LIN {X 0,Y 639.897,Z 1293.567,A -85,B 0,C 180,E1 29787.314,E2 29787.314} C_VEL
LIN {X 0,Y 639.907,Z 1290.691,A -85,B 0,C 180,E1 29785.251,E2 29785.251} C_VEL
LIN {X 0,Y 639.948,Z 1285.814,A -85,B 0,C 180,E1 29783.091,E2 29783.091} C_VEL
LIN {X 0,Y 640.038,Z 1280.646,A -85,B 0,C 180,E1 29781.376,E2 29781.376} C_VEL
LIN {X 0,Y 640.175,Z 1274.233,A -85,B 0,C 180,E1 29779.654,E2 29779.654} C_VEL
LIN {X 0,Y 640.418,Z 1265.861,A -85,B 0,C 180,E1 29777.791,E2 29777.791} C_VEL
LIN {X 0,Y 640.846,Z 1254.401,A -85,B 0,C 180,E1 29775.68,E2 29775.68} C_VEL
LIN {X 0,Y 641.338,Z 1242.79,A -85,B 0,C 180,E1 29773.89,E2 29773.89} C_VEL
LIN {X 0,Y 641.901,Z 1231.865,A -85,B 0,C 180,E1 29772.412,E2 29772.412} C_VEL
LIN {X 0,Y 642.587,Z 1219.47,A -85,B 0,C 180,E1 29770.929,E2 29770.929} C_VEL
LIN {X 0,Y 643.506,Z 1204.493,A -85,B 0,C 180,E1 29769.348,E2 29769.348} C_VEL
LIN {X 0,Y 644.672,Z 1186.015,A -85,B 0,C 180,E1 29767.668,E2 29767.668} C_VEL
LIN {X 0,Y 645.836,Z 1168.25,A -85,B 0,C 180,E1 29766.265,E2 29766.265} C_VEL
LIN {X 0,Y 647.147,Z 1148.227,A -85,B 0,C 180,E1 29764.907,E2 29764.907} C_VEL
LIN {X 0,Y 648.4,Z 1127.933,A -85,B 0,C 180,E1 29763.733,E2 29763.733} C_VEL
LIN {X 0,Y 649.554,Z 1106.2,A -85,B 0,C 180,E1 29762.697,E2 29762.697} C_VEL
LIN {X 0,Y 650.662,Z 1083.667,A -85,B 0,C 180,E1 29761.802,E2 29761.802} C_VEL
LIN {X 0,Y 651.674,Z 1060.243,A -85,B 0,C 180,E1 29761.049,E2 29761.049} C_VEL
LIN {X 0,Y 652.617,Z 1036.441,A -85,B 0,C 180,E1 29760.454,E2 29760.454} C_VEL
LIN {X 0,Y 653.293,Z 1013.421,A -85,B 0,C 180,E1 29760.036,E2 29760.036} C_VEL
LIN {X 0,Y 654.171,Z 971.336,A -85,B 0,C 180,E1 29759.507,E2 29759.507} C_VEL
LIN {X 0,Y 659.659,Z 959.553,A -85,B 0,C 180,E1 29758.879,E2 29758.879} C_VEL
LIN {X 0,Y 664.536,Z 951.202,A -85,B 0,C 180,E1 29758.477,E2 29758.477} C_VEL
LIN {X 0,Y 670.603,Z 941.643,A -85,B 0,C 180,E1 29758.043,E2 29758.043} C_VEL
LIN {X 0,Y 679.475,Z 930.778,A -85,B 0,C 180,E1 29757.638,E2 29757.638} C_VEL
LIN {X 0,Y 692.272,Z 917.65,A -85,B 0,C 180,E1 29757.261,E2 29757.261} C_VEL
LIN {X 0,Y 701.55,Z 907.268,A -85,B 0,C 180,E1 29757.112,E2 29757.112} C_VEL
LIN {X 0,Y 709.193,Z 894.911,A -85,B 0,C 180,E1 29756.838,E2 29756.838} C_VEL
LIN {X 0,Y 716.952,Z 880.627,A -85,B 0,C 180,E1 29756.657,E2 29756.657} C_VEL
LIN {X 0,Y 714.524,Z 882.399,A -85,B 0,C 180,E1 29756.226,E2 29756.226} C_VEL
LIN {X 0,Y 710.853,Z 883.16,A -85,B 0,C 180,E1 29755.801,E2 29755.801} C_VEL
LIN {X 0,Y 705.825,Z 882.559,A -85,B 0,C 180,E1 29755.393,E2 29755.393} C_VEL
LIN {X 0,Y 694.35,Z 878.529,A -85,B 0,C 180,E1 29754.594,E2 29754.594} C_VEL
LIN {X 0,Y 684.4,Z 873.303,A -85,B 0,C 180,E1 29753.752,E2 29753.752} C_VEL
LIN {X 0,Y 675.328,Z 866.486,A -85,B 0,C 180,E1 29752.803,E2 29752.803} C_VEL
LIN {X 0,Y 667.782,Z 858.379,A -85,B 0,C 180,E1 29751.803,E2 29751.803} C_VEL
LIN {X 0,Y 661.627,Z 848.569,A -85,B 0,C 180,E1 29750.714,E2 29750.714} C_VEL
LIN {X 0,Y 657.041,Z 836.989,A -85,B 0,C 180,E1 29749.544,E2 29749.544} C_VEL
LIN {X 0,Y 654.419,Z 824.683,A -85,B 0,C 180,E1 29748.41,E2 29748.41} C_VEL
LIN {X 0,Y 653.38,Z 808.168,A -85,B 0,C 180,E1 29747.013,E2 29747.013} C_VEL
LIN {X 0,Y 655.589,Z 761.985,A -85,B 0,C 180,E1 29743.341,E2 29743.341} C_VEL
LIN {X 0,Y 657.511,Z 726.256,A -85,B 0,C 180,E1 29740.43,E2 29740.43} C_VEL
LIN {X 0,Y 659.372,Z 691.646,A -85,B 0,C 180,E1 29737.528,E2 29737.528} C_VEL
LIN {X 0,Y 661.157,Z 657.905,A -85,B 0,C 180,E1 29734.608,E2 29734.608} C_VEL
LIN {X 0,Y 661.133,Z 654.991,A -85,B 0,C 180,E1 29734.337,E2 29734.337} C_VEL
LIN {X 0,Y 652.452,Z 634.727,A -85,B 0,C 180,E1 29731.609,E2 29731.609} C_VEL
LIN {X 0,Y 645.602,Z 619.347,A -85,B 0,C 180,E1 29729.404,E2 29729.404} C_VEL
LIN {X 0,Y 642.088,Z 611.595,A -85,B 0,C 180,E1 29728.256,E2 29728.256} C_VEL
LIN {X 0,Y 640.822,Z 608.156,A -85,B 0,C 180,E1 29727.737,E2 29727.737} C_VEL
LIN {X 0,Y 640.824,Z 608.157,A -85,B 0,C 180,E1 29724.621,E2 29724.621} C_VEL
LIN {X 0,Y 640.829,Z 608.159,A -85,B 0,C 180,E1 29721.415,E2 29721.415} C_VEL
LIN {X 0,Y 640.828,Z 608.156,A -85,B 0,C 180,E1 29718.278,E2 29718.278} C_VEL
LIN {X 0,Y 640.832,Z 608.155,A -85,B 0,C 180,E1 29715.03,E2 29715.03} C_VEL
LIN {X 0,Y 640.836,Z 608.156,A -85,B 0,C 180,E1 29711.886,E2 29711.886} C_VEL
LIN {X 0,Y 640.828,Z 608.156,A -85,B 0,C 180,E1 29708.705,E2 29708.705} C_VEL
LIN {X 0,Y 640.835,Z 608.152,A -85,B 0,C 180,E1 29705.551,E2 29705.551} C_VEL
LIN {X 0,Y 640.822,Z 608.159,A -85,B 0,C 180,E1 29702.325,E2 29702.325} C_VEL
LIN {X 0,Y 640.833,Z 608.158,A -85,B 0,C 180,E1 29699.195,E2 29699.195} C_VEL
LIN {X 0,Y 640.819,Z 608.158,A -85,B 0,C 180,E1 29696.063,E2 29696.063} C_VEL
LIN {X 0,Y 640.828,Z 608.156,A -85,B 0,C 180,E1 29692.895,E2 29692.895} C_VEL
LIN {X 0,Y 640.816,Z 608.156,A -85,B 0,C 180,E1 29689.754,E2 29689.754} C_VEL
LIN {X 0,Y 640.823,Z 608.154,A -85,B 0,C 180,E1 29686.648,E2 29686.648} C_VEL
LIN {X 0,Y 640.817,Z 608.154,A -85,B 0,C 180,E1 29683.595,E2 29683.595} C_VEL
LIN {X 0,Y 640.823,Z 608.154,A -85,B 0,C 180,E1 29680.458,E2 29680.458} C_VEL
LIN {X 0,Y 640.816,Z 608.156,A -85,B 0,C 180,E1 29677.331,E2 29677.331} C_VEL
LIN {X 0,Y 640.818,Z 608.156,A -85,B 0,C 180,E1 29674.193,E2 29674.193} C_VEL
LIN {X 0,Y 640.816,Z 608.156,A -85,B 0,C 180,E1 29671.082,E2 29671.082} C_VEL
LIN {X 0,Y 640.816,Z 608.155,A -85,B 0,C 180,E1 29667.96,E2 29667.96} C_VEL
LIN {X 0,Y 640.815,Z 608.151,A -85,B 0,C 180,E1 29664.844,E2 29664.844} C_VEL
LIN {X 0,Y 640.816,Z 608.152,A -85,B 0,C 180,E1 29661.723,E2 29661.723} C_VEL
LIN {X 0,Y 640.817,Z 608.154,A -85,B 0,C 180,E1 29658.633,E2 29658.633} C_VEL
LIN {X 0,Y 640.817,Z 608.152,A -85,B 0,C 180,E1 29655.483,E2 29655.483} C_VEL
LIN {X 0,Y 640.832,Z 608.158,A -85,B 0,C 180,E1 29654.378,E2 29654.378} C_VEL
LIN {X 0,Y 639.852,Z 608.286,A -85,B 0,C 180,E1 29653.69,E2 29653.69} C_VEL
LIN {X 0,Y 633.444,Z 609.065,A -85,B 0,C 180,E1 29651.759,E2 29651.759} C_VEL
LIN {X 0,Y 632.89,Z 609.134,A -85,B 0,C 180,E1 29651.257,E2 29651.257} C_VEL
LIN {X 0,Y 632.886,Z 609.141,A -85,B 0,C 180,E1 29648.114,E2 29648.114} C_VEL
LIN {X 0,Y 632.892,Z 609.141,A -85,B 0,C 180,E1 29644.919,E2 29644.919} C_VEL
LIN {X 0,Y 632.906,Z 609.283,A -85,B 0,C 180,E1 29642.246,E2 29642.246} C_VEL
LIN {X 0,Y 640.506,Z 633.883,A -85,B 0,C 180,E1 29640.279,E2 29640.279} C_VEL
LIN {X 0,Y 639.937,Z 670.595,A -85,B 0,C 180,E1 29637.804,E2 29637.804} C_VEL
LIN {X 0,Y 638.884,Z 712.937,A -85,B 0,C 180,E1 29634.896,E2 29634.896} C_VEL
LIN {X 0,Y 637.709,Z 757.785,A -85,B 0,C 180,E1 29631.813,E2 29631.813} C_VEL
LIN {X 0,Y 636.616,Z 804.939,A -85,B 0,C 180,E1 29628.639,E2 29628.639} C_VEL
LIN {X 0,Y 636.165,Z 836.355,A -85,B 0,C 180,E1 29626.604,E2 29626.604} C_VEL
LIN {X 0,Y 636.961,Z 845.526,A -85,B 0,C 180,E1 29626.473,E2 29626.473} C_VEL
LIN {X 0,Y 635.944,Z 1005.419,A -85,B 0,C 180,E1 29624.624,E2 29624.624} C_VEL
LIN {X 0,Y 635.746,Z 1022.874,A -85,B 0,C 180,E1 29624.256,E2 29624.256} C_VEL
LIN {X 0,Y 635.419,Z 1039.147,A -85,B 0,C 180,E1 29623.744,E2 29623.744} C_VEL
LIN {X 0,Y 634.987,Z 1055.365,A -85,B 0,C 180,E1 29623.058,E2 29623.058} C_VEL
LIN {X 0,Y 634.509,Z 1070.531,A -85,B 0,C 180,E1 29622.235,E2 29622.235} C_VEL
LIN {X 0,Y 634.009,Z 1084.629,A -85,B 0,C 180,E1 29621.276,E2 29621.276} C_VEL
LIN {X 0,Y 633.52,Z 1097.632,A -85,B 0,C 180,E1 29620.18,E2 29620.18} C_VEL
LIN {X 0,Y 633.087,Z 1109.143,A -85,B 0,C 180,E1 29618.994,E2 29618.994} C_VEL
LIN {X 0,Y 632.73,Z 1119.243,A -85,B 0,C 180,E1 29617.718,E2 29617.718} C_VEL
LIN {X 0,Y 632.454,Z 1127.914,A -85,B 0,C 180,E1 29616.352,E2 29616.352} C_VEL
LIN {X 0,Y 632.266,Z 1135.129,A -85,B 0,C 180,E1 29614.898,E2 29614.898} C_VEL
LIN {X 0,Y 632.152,Z 1140.845,A -85,B 0,C 180,E1 29613.354,E2 29613.354} C_VEL
LIN {X 0,Y 632.086,Z 1144.759,A -85,B 0,C 180,E1 29611.812,E2 29611.812} C_VEL
LIN {X 0,Y 632.068,Z 1147.012,A -85,B 0,C 180,E1 29610.18,E2 29610.18} C_VEL
LIN {X 0,Y 632.054,Z 1147.461,A -85,B 0,C 180,E1 29608.548,E2 29608.548} C_VEL
LIN {X 0,Y 632.072,Z 1146.132,A -85,B 0,C 180,E1 29606.916,E2 29606.916} C_VEL
LIN {X 0,Y 632.113,Z 1143.147,A -85,B 0,C 180,E1 29605.372,E2 29605.372} C_VEL
LIN {X 0,Y 632.203,Z 1138.378,A -85,B 0,C 180,E1 29603.825,E2 29603.825} C_VEL
LIN {X 0,Y 632.352,Z 1131.721,A -85,B 0,C 180,E1 29602.275,E2 29602.275} C_VEL
LIN {X 0,Y 632.597,Z 1123.458,A -85,B 0,C 180,E1 29600.813,E2 29600.813} C_VEL
LIN {X 0,Y 632.926,Z 1113.551,A -85,B 0,C 180,E1 29599.439,E2 29599.439} C_VEL
LIN {X 0,Y 633.356,Z 1102.074,A -85,B 0,C 180,E1 29598.156,E2 29598.156} C_VEL
LIN {X 0,Y 633.841,Z 1089.419,A -85,B 0,C 180,E1 29597.008,E2 29597.008} C_VEL
LIN {X 0,Y 634.337,Z 1075.597,A -85,B 0,C 180,E1 29595.997,E2 29595.997} C_VEL
LIN {X 0,Y 634.847,Z 1060.153,A -85,B 0,C 180,E1 29595.089,E2 29595.089} C_VEL
LIN {X 0,Y 635.28,Z 1044.944,A -85,B 0,C 180,E1 29594.386,E2 29594.386} C_VEL
LIN {X 0,Y 635.649,Z 1028.193,A -85,B 0,C 180,E1 29593.804,E2 29593.804} C_VEL
LIN {X 0,Y 635.902,Z 1010.504,A -85,B 0,C 180,E1 29593.376,E2 29593.376} C_VEL
LIN {X 0,Y 636.039,Z 990.987,A -85,B 0,C 180,E1 29593.097,E2 29593.097} C_VEL
LIN {X 0,Y 636.768,Z 841.145,A -85,B 0,C 180,E1 29591.38,E2 29591.38} C_VEL
LIN {X 0,Y 636.079,Z 835.695,A -85,B 0,C 180,E1 29591.295,E2 29591.295} C_VEL
LIN {X 0,Y 637.03,Z 786.131,A -85,B 0,C 180,E1 29588.015,E2 29588.015} C_VEL
LIN {X 0,Y 638.19,Z 740.132,A -85,B 0,C 180,E1 29584.874,E2 29584.874} C_VEL
LIN {X 0,Y 639.395,Z 696.862,A -85,B 0,C 180,E1 29581.884,E2 29581.884} C_VEL
LIN {X 0,Y 640.369,Z 654.586,A -85,B 0,C 180,E1 29578.984,E2 29578.984} C_VEL
LIN {X 0,Y 640.439,Z 633.256,A -85,B 0,C 180,E1 29577.542,E2 29577.542} C_VEL
LIN {X 0,Y 632.885,Z 609.139,A -85,B 0,C 180,E1 29575.559,E2 29575.559} C_VEL
LIN {X 0,Y 632.882,Z 609.145,A -85,B 0,C 180,E1 29572.329,E2 29572.329} C_VEL
LIN {X 0,Y 632.896,Z 609.135,A -85,B 0,C 180,E1 29569.15,E2 29569.15} C_VEL
LIN {X 0,Y 632.877,Z 609.144,A -85,B 0,C 180,E1 29565.959,E2 29565.959} C_VEL
LIN {X 0,Y 632.876,Z 609.144,A -85,B 0,C 180,E1 29562.854,E2 29562.854} C_VEL
LIN {X 0,Y 632.89,Z 609.145,A -85,B 0,C 180,E1 29559.781,E2 29559.781} C_VEL
LIN {X 0,Y 632.879,Z 609.146,A -85,B 0,C 180,E1 29556.621,E2 29556.621} C_VEL
LIN {X 0,Y 632.891,Z 609.15,A -85,B 0,C 180,E1 29553.462,E2 29553.462} C_VEL
LIN {X 0,Y 632.915,Z 609.376,A -85,B 0,C 180,E1 29552.998,E2 29552.998} C_VEL
LIN {X 0,Y 634.657,Z 613.86,A -85,B 0,C 180,E1 29552.448,E2 29552.448} C_VEL
LIN {X 0,Y 644.095,Z 628.518,A -85,B 0,C 180,E1 29551.604,E2 29551.604} C_VEL
LIN {X 0,Y 650.556,Z 639.812,A -85,B 0,C 180,E1 29551.027,E2 29551.027} C_VEL
LIN {X 0,Y 648.075,Z 791.876,A -85,B 0,C 180,E1 29549.096,E2 29549.096} C_VEL
LIN {X 0,Y 646.526,Z 902.715,A -85,B 0,C 180,E1 29547.714,E2 29547.714} C_VEL
LIN {X 0,Y 645.796,Z 953.532,A -85,B 0,C 180,E1 29547.058,E2 29547.058} C_VEL
LIN {X 0,Y 645.049,Z 977.906,A -85,B 0,C 180,E1 29546.565,E2 29546.565} C_VEL
LIN {X 0,Y 644.199,Z 999.937,A -85,B 0,C 180,E1 29545.958,E2 29545.958} C_VEL
LIN {X 0,Y 643.14,Z 1022.537,A -85,B 0,C 180,E1 29545.169,E2 29545.169} C_VEL
LIN {X 0,Y 641.904,Z 1044.009,A -85,B 0,C 180,E1 29544.233,E2 29544.233} C_VEL
LIN {X 0,Y 640.848,Z 1061.28,A -85,B 0,C 180,E1 29543.348,E2 29543.348} C_VEL
LIN {X 0,Y 639.771,Z 1077.595,A -85,B 0,C 180,E1 29542.387,E2 29542.387} C_VEL
LIN {X 0,Y 638.664,Z 1093.449,A -85,B 0,C 180,E1 29541.324,E2 29541.324} C_VEL
LIN {X 0,Y 637.522,Z 1109.728,A -85,B 0,C 180,E1 29540.089,E2 29540.089} C_VEL
LIN {X 0,Y 636.21,Z 1128.852,A -85,B 0,C 180,E1 29538.415,E2 29538.415} C_VEL
LIN {X 0,Y 635.223,Z 1143.488,A -85,B 0,C 180,E1 29536.93,E2 29536.93} C_VEL
LIN {X 0,Y 634.46,Z 1155.662,A -85,B 0,C 180,E1 29535.54,E2 29535.54} C_VEL
LIN {X 0,Y 633.782,Z 1167.178,A -85,B 0,C 180,E1 29534.061,E2 29534.061} C_VEL
LIN {X 0,Y 633.229,Z 1177.944,A -85,B 0,C 180,E1 29532.494,E2 29532.494} C_VEL
LIN {X 0,Y 632.78,Z 1187.36,A -85,B 0,C 180,E1 29530.931,E2 29530.931} C_VEL
LIN {X 0,Y 632.476,Z 1195.561,A -85,B 0,C 180,E1 29529.372,E2 29529.372} C_VEL
LIN {X 0,Y 632.221,Z 1203.41,A -85,B 0,C 180,E1 29527.634,E2 29527.634} C_VEL
LIN {X 0,Y 632.047,Z 1210.905,A -85,B 0,C 180,E1 29525.629,E2 29525.629} C_VEL
LIN {X 0,Y 631.95,Z 1217.313,A -85,B 0,C 180,E1 29523.356,E2 29523.356} C_VEL
LIN {X 0,Y 631.916,Z 1221.027,A -85,B 0,C 180,E1 29521.541,E2 29521.541} C_VEL
LIN {X 0,Y 631.906,Z 1223.496,A -85,B 0,C 180,E1 29519.728,E2 29519.728} C_VEL
LIN {X 0,Y 631.908,Z 1224.737,A -85,B 0,C 180,E1 29517.914,E2 29517.914} C_VEL
LIN {X 0,Y 631.914,Z 1224.788,A -85,B 0,C 180,E1 29516.189,E2 29516.189} C_VEL
LIN {X 0,Y 631.912,Z 1223.741,A -85,B 0,C 180,E1 29514.436,E2 29514.436} C_VEL
LIN {X 0,Y 631.921,Z 1221.197,A -85,B 0,C 180,E1 29512.453,E2 29512.453} C_VEL
LIN {X 0,Y 631.966,Z 1216.378,A -85,B 0,C 180,E1 29510.161,E2 29510.161} C_VEL
LIN {X 0,Y 632.052,Z 1210.665,A -85,B 0,C 180,E1 29508.225,E2 29508.225} C_VEL
LIN {X 0,Y 632.205,Z 1204.172,A -85,B 0,C 180,E1 29506.463,E2 29506.463} C_VEL
LIN {X 0,Y 632.439,Z 1196.31,A -85,B 0,C 180,E1 29504.691,E2 29504.691} C_VEL
LIN {X 0,Y 632.785,Z 1187.497,A -85,B 0,C 180,E1 29503.003,E2 29503.003} C_VEL
LIN {X 0,Y 633.295,Z 1176.659,A -85,B 0,C 180,E1 29501.211,E2 29501.211} C_VEL
LIN {X 0,Y 634.06,Z 1162.49,A -85,B 0,C 180,E1 29499.218,E2 29499.218} C_VEL
LIN {X 0,Y 634.861,Z 1149.049,A -85,B 0,C 180,E1 29497.595,E2 29497.595} C_VEL
LIN {X 0,Y 635.713,Z 1136.053,A -85,B 0,C 180,E1 29496.206,E2 29496.206} C_VEL
LIN {X 0,Y 636.625,Z 1122.428,A -85,B 0,C 180,E1 29494.908,E2 29494.908} C_VEL
LIN {X 0,Y 637.619,Z 1108.234,A -85,B 0,C 180,E1 29493.704,E2 29493.704} C_VEL
LIN {X 0,Y 638.659,Z 1093.556,A -85,B 0,C 180,E1 29492.594,E2 29492.594} C_VEL
LIN {X 0,Y 639.621,Z 1079.005,A -85,B 0,C 180,E1 29491.626,E2 29491.626} C_VEL
LIN {X 0,Y 640.712,Z 1061.526,A -85,B 0,C 180,E1 29490.606,E2 29490.606} C_VEL
LIN {X 0,Y 641.904,Z 1039.745,A -85,B 0,C 180,E1 29489.534,E2 29489.534} C_VEL
LIN {X 0,Y 642.868,Z 1018.864,A -85,B 0,C 180,E1 29488.702,E2 29488.702} C_VEL
LIN {X 0,Y 643.612,Z 999.264,A -85,B 0,C 180,E1 29488.058,E2 29488.058} C_VEL
LIN {X 0,Y 644.271,Z 976.224,A -85,B 0,C 180,E1 29487.472,E2 29487.472} C_VEL
LIN {X 0,Y 644.765,Z 952.724,A -85,B 0,C 180,E1 29487.047,E2 29487.047} C_VEL
LIN {X 0,Y 645.24,Z 868.019,A -85,B 0,C 180,E1 29486.099,E2 29486.099} C_VEL
LIN {X 0,Y 646.392,Z 666.407,A -85,B 0,C 180,E1 29483.836,E2 29483.836} C_VEL
LIN {X 0,Y 646.514,Z 638.485,A -85,B 0,C 180,E1 29483.499,E2 29483.499} C_VEL
LIN {X 0,Y 643.79,Z 635.766,A -85,B 0,C 180,E1 29483.341,E2 29483.341} C_VEL
LIN {X 0,Y 644,Z 636.198,A -85,B 0,C 180,E1 29482.172,E2 29482.172} C_VEL
LIN {X 0,Y 644.603,Z 638.016,A -85,B 0,C 180,E1 29481.195,E2 29481.195} C_VEL
LIN {X 0,Y 645.736,Z 641.08,A -85,B 0,C 180,E1 29480.178,E2 29480.178} C_VEL
LIN {X 0,Y 645.925,Z 642.037,A -85,B 0,C 180,E1 29479.951,E2 29479.951} C_VEL
LIN {X 0,Y 641.41,Z 653.382,A -85,B 0,C 180,E1 29478.712,E2 29478.712} C_VEL
LIN {X 0,Y 638.172,Z 666.32,A -85,B 0,C 180,E1 29477.523,E2 29477.523} C_VEL
LIN {X 0,Y 635.905,Z 681.652,A -85,B 0,C 180,E1 29476.328,E2 29476.328} C_VEL
LIN {X 0,Y 634.23,Z 702.463,A -85,B 0,C 180,E1 29474.935,E2 29474.935} C_VEL
LIN {X 0,Y 633.019,Z 734.797,A -85,B 0,C 180,E1 29473.03,E2 29473.03} C_VEL
LIN {X 0,Y 632.986,Z 773.811,A -85,B 0,C 180,E1 29470.88,E2 29470.88} C_VEL
LIN {X 0,Y 634.85,Z 794.261,A -85,B 0,C 180,E1 29469.752,E2 29469.752} C_VEL
LIN {X 0,Y 638.194,Z 811.119,A -85,B 0,C 180,E1 29468.808,E2 29468.808} C_VEL
LIN {X 0,Y 643.087,Z 825.935,A -85,B 0,C 180,E1 29467.973,E2 29467.973} C_VEL
LIN {X 0,Y 649.932,Z 840.295,A -85,B 0,C 180,E1 29467.163,E2 29467.163} C_VEL
LIN {X 0,Y 657.821,Z 852.497,A -85,B 0,C 180,E1 29466.478,E2 29466.478} C_VEL
LIN {X 0,Y 667.384,Z 863.872,A -85,B 0,C 180,E1 29465.851,E2 29465.851} C_VEL
LIN {X 0,Y 678.649,Z 874.385,A -85,B 0,C 180,E1 29465.29,E2 29465.29} C_VEL
LIN {X 0,Y 690.663,Z 883.187,A -85,B 0,C 180,E1 29464.829,E2 29464.829} C_VEL
LIN {X 0,Y 697.221,Z 887.009,A -85,B 0,C 180,E1 29464.595,E2 29464.595} C_VEL
LIN {X 0,Y 702.925,Z 889.045,A -85,B 0,C 180,E1 29464.285,E2 29464.285} C_VEL
LIN {X 0,Y 707.445,Z 889.627,A -85,B 0,C 180,E1 29463.936,E2 29463.936} C_VEL
LIN {X 0,Y 708.595,Z 889.733,A -85,B 0,C 180,E1 29463.813,E2 29463.813} C_VEL
LIN {X 0,Y 699.671,Z 901.616,A -85,B 0,C 180,E1 29463.529,E2 29463.529} C_VEL
LIN {X 0,Y 696.631,Z 905.632,A -85,B 0,C 180,E1 29463.398,E2 29463.398} C_VEL
LIN {X 0,Y 686.664,Z 914.581,A -85,B 0,C 180,E1 29463.144,E2 29463.144} C_VEL
LIN {X 0,Y 675.161,Z 924.295,A -85,B 0,C 180,E1 29462.672,E2 29462.672} C_VEL
LIN {X 0,Y 665.009,Z 934.556,A -85,B 0,C 180,E1 29462.109,E2 29462.109} C_VEL
LIN {X 0,Y 657.922,Z 944.123,A -85,B 0,C 180,E1 29461.572,E2 29461.572} C_VEL
LIN {X 0,Y 649.022,Z 959.216,A -85,B 0,C 180,E1 29460.712,E2 29460.712} C_VEL
LIN {X 0,Y 646.755,Z 964.415,A -85,B 0,C 180,E1 29460.447,E2 29460.447} C_VEL
LIN {X 0,Y 644.912,Z 973.272,A -85,B 0,C 180,E1 29460.398,E2 29460.398} C_VEL
LIN {X 0,Y 644.423,Z 1012.046,A -85,B 0,C 180,E1 29459.935,E2 29459.935} C_VEL
LIN {X 0,Y 643.83,Z 1038.212,A -85,B 0,C 180,E1 29459.462,E2 29459.462} C_VEL
LIN {X 0,Y 643.11,Z 1062.478,A -85,B 0,C 180,E1 29458.87,E2 29458.87} C_VEL
LIN {X 0,Y 642.378,Z 1085.145,A -85,B 0,C 180,E1 29458.177,E2 29458.177} C_VEL
LIN {X 0,Y 641.485,Z 1108.187,A -85,B 0,C 180,E1 29457.318,E2 29457.318} C_VEL
LIN {X 0,Y 640.506,Z 1130.491,A -85,B 0,C 180,E1 29456.319,E2 29456.319} C_VEL
LIN {X 0,Y 639.636,Z 1148.325,A -85,B 0,C 180,E1 29455.362,E2 29455.362} C_VEL
LIN {X 0,Y 638.63,Z 1164.294,A -85,B 0,C 180,E1 29454.317,E2 29454.317} C_VEL
LIN {X 0,Y 637.434,Z 1180.844,A -85,B 0,C 180,E1 29453.041,E2 29453.041} C_VEL
LIN {X 0,Y 636.455,Z 1195.131,A -85,B 0,C 180,E1 29451.8,E2 29451.8} C_VEL
LIN {X 0,Y 635.575,Z 1208.117,A -85,B 0,C 180,E1 29450.539,E2 29450.539} C_VEL
LIN {X 0,Y 634.734,Z 1221.071,A -85,B 0,C 180,E1 29449.128,E2 29449.128} C_VEL
LIN {X 0,Y 634.009,Z 1233.284,A -85,B 0,C 180,E1 29447.627,E2 29447.627} C_VEL
LIN {X 0,Y 633.349,Z 1245.331,A -85,B 0,C 180,E1 29445.945,E2 29445.945} C_VEL
LIN {X 0,Y 632.753,Z 1258.357,A -85,B 0,C 180,E1 29443.806,E2 29443.806} C_VEL
LIN {X 0,Y 632.418,Z 1267.357,A -85,B 0,C 180,E1 29442.047,E2 29442.047} C_VEL
LIN {X 0,Y 632.181,Z 1274.952,A -85,B 0,C 180,E1 29440.297,E2 29440.297} C_VEL
LIN {X 0,Y 632.044,Z 1281.234,A -85,B 0,C 180,E1 29438.553,E2 29438.553} C_VEL
LIN {X 0,Y 631.951,Z 1287.265,A -85,B 0,C 180,E1 29436.451,E2 29436.451} C_VEL
LIN {X 0,Y 631.913,Z 1291.566,A -85,B 0,C 180,E1 29434.266,E2 29434.266} C_VEL
LIN {X 0,Y 631.901,Z 1293.89,A -85,B 0,C 180,E1 29432.359,E2 29432.359} C_VEL
LIN {X 0,Y 631.893,Z 1294.865,A -85,B 0,C 180,E1 29430.545,E2 29430.545} C_VEL
LIN {X 0,Y 631.892,Z 1294.559,A -85,B 0,C 180,E1 29428.46,E2 29428.46} C_VEL
LIN {X 0,Y 631.9,Z 1292.387,A -85,B 0,C 180,E1 29426.282,E2 29426.282} C_VEL
LIN {X 0,Y 631.921,Z 1289.037,A -85,B 0,C 180,E1 29424.371,E2 29424.371} C_VEL
LIN {X 0,Y 631.991,Z 1284.804,A -85,B 0,C 180,E1 29422.639,E2 29422.639} C_VEL
LIN {X 0,Y 632.068,Z 1279.397,A -85,B 0,C 180,E1 29420.899,E2 29420.899} C_VEL
LIN {X 0,Y 632.276,Z 1271.619,A -85,B 0,C 180,E1 29418.877,E2 29418.877} C_VEL
LIN {X 0,Y 632.632,Z 1261.37,A -85,B 0,C 180,E1 29416.753,E2 29416.753} C_VEL
LIN {X 0,Y 633.026,Z 1251.836,A -85,B 0,C 180,E1 29415.082,E2 29415.082} C_VEL
LIN {X 0,Y 633.521,Z 1242.136,A -85,B 0,C 180,E1 29413.591,E2 29413.591} C_VEL
LIN {X 0,Y 634.13,Z 1231.127,A -85,B 0,C 180,E1 29412.094,E2 29412.094} C_VEL
LIN {X 0,Y 634.895,Z 1218.644,A -85,B 0,C 180,E1 29410.593,E2 29410.593} C_VEL
LIN {X 0,Y 635.991,Z 1202.167,A -85,B 0,C 180,E1 29408.851,E2 29408.851} C_VEL
LIN {X 0,Y 637.169,Z 1184.867,A -85,B 0,C 180,E1 29407.293,E2 29407.293} C_VEL
LIN {X 0,Y 638.369,Z 1167.956,A -85,B 0,C 180,E1 29405.947,E2 29405.947} C_VEL
LIN {X 0,Y 639.448,Z 1151.512,A -85,B 0,C 180,E1 29404.831,E2 29404.831} C_VEL
LIN {X 0,Y 640.748,Z 1130.264,A -85,B 0,C 180,E1 29403.595,E2 29403.595} C_VEL
LIN {X 0,Y 642.017,Z 1108.247,A -85,B 0,C 180,E1 29402.506,E2 29402.506} C_VEL
LIN {X 0,Y 643.29,Z 1085.07,A -85,B 0,C 180,E1 29401.553,E2 29401.553} C_VEL
LIN {X 0,Y 644.468,Z 1060.94,A -85,B 0,C 180,E1 29400.748,E2 29400.748} C_VEL
LIN {X 0,Y 645.547,Z 1036.841,A -85,B 0,C 180,E1 29400.124,E2 29400.124} C_VEL
LIN {X 0,Y 646.347,Z 1013.026,A -85,B 0,C 180,E1 29399.678,E2 29399.678} C_VEL
LIN {X 0,Y 647.327,Z 970.69,A -85,B 0,C 180,E1 29399.145,E2 29399.145} C_VEL
LIN {X 0,Y 647.893,Z 968.867,A -85,B 0,C 180,E1 29399.077,E2 29399.077} C_VEL
LIN {X 0,Y 653.309,Z 957.677,A -85,B 0,C 180,E1 29398.484,E2 29398.484} C_VEL
LIN {X 0,Y 662.94,Z 941.728,A -85,B 0,C 180,E1 29397.731,E2 29397.731} C_VEL
LIN {X 0,Y 671.242,Z 931.043,A -85,B 0,C 180,E1 29397.313,E2 29397.313} C_VEL
LIN {X 0,Y 683.251,Z 918.336,A -85,B 0,C 180,E1 29396.919,E2 29396.919} C_VEL
LIN {X 0,Y 697.669,Z 904.35,A -85,B 0,C 180,E1 29396.562,E2 29396.562} C_VEL
LIN {X 0,Y 706.24,Z 892.92,A -85,B 0,C 180,E1 29396.248,E2 29396.248} C_VEL
LIN {X 0,Y 708.556,Z 889.584,A -85,B 0,C 180,E1 29396.169,E2 29396.169} C_VEL
LIN {X 0,Y 703.814,Z 889.238,A -85,B 0,C 180,E1 29395.775,E2 29395.775} C_VEL
LIN {X 0,Y 691.427,Z 885.234,A -85,B 0,C 180,E1 29394.936,E2 29394.936} C_VEL
LIN {X 0,Y 680.59,Z 879.9,A -85,B 0,C 180,E1 29394.048,E2 29394.048} C_VEL
LIN {X 0,Y 670.686,Z 872.883,A -85,B 0,C 180,E1 29393.044,E2 29393.044} C_VEL
LIN {X 0,Y 662.472,Z 864.527,A -85,B 0,C 180,E1 29391.987,E2 29391.987} C_VEL
LIN {X 0,Y 656.416,Z 855.68,A -85,B 0,C 180,E1 29390.974,E2 29390.974} C_VEL
LIN {X 0,Y 651.308,Z 844.456,A -85,B 0,C 180,E1 29389.798,E2 29389.798} C_VEL
LIN {X 0,Y 647.974,Z 831.785,A -85,B 0,C 180,E1 29388.586,E2 29388.586} C_VEL
LIN {X 0,Y 646.455,Z 816.908,A -85,B 0,C 180,E1 29387.282,E2 29387.282} C_VEL
LIN {X 0,Y 646.864,Z 797.203,A -85,B 0,C 180,E1 29385.681,E2 29385.681} C_VEL
LIN {X 0,Y 648.952,Z 759.88,A -85,B 0,C 180,E1 29382.683,E2 29382.683} C_VEL
LIN {X 0,Y 650.979,Z 724.578,A -85,B 0,C 180,E1 29379.778,E2 29379.778} C_VEL
LIN {X 0,Y 652.917,Z 690.527,A -85,B 0,C 180,E1 29376.893,E2 29376.893} C_VEL
LIN {X 0,Y 654.678,Z 659.351,A -85,B 0,C 180,E1 29374.169,E2 29374.169} C_VEL
LIN {X 0,Y 646.087,Z 639.23,A -85,B 0,C 180,E1 29371.436,E2 29371.436} C_VEL
LIN {X 0,Y 638.251,Z 621.301,A -85,B 0,C 180,E1 29368.85,E2 29368.85} C_VEL
LIN {X 0,Y 634.191,Z 612.62,A -85,B 0,C 180,E1 29367.514,E2 29367.514} C_VEL
LIN {X 0,Y 632.878,Z 609.148,A -85,B 0,C 180,E1 29366.964,E2 29366.964} C_VEL
LIN {X 0,Y 632.874,Z 609.148,A -85,B 0,C 180,E1 29363.831,E2 29363.831} C_VEL
LIN {X 0,Y 632.882,Z 609.144,A -85,B 0,C 180,E1 29360.823,E2 29360.823} C_VEL
LIN {X 0,Y 632.875,Z 609.147,A -85,B 0,C 180,E1 29357.701,E2 29357.701} C_VEL
LIN {X 0,Y 632.892,Z 609.145,A -85,B 0,C 180,E1 29354.642,E2 29354.642} C_VEL
LIN {X 0,Y 632.881,Z 609.146,A -85,B 0,C 180,E1 29351.482,E2 29351.482} C_VEL
LIN {X 0,Y 632.894,Z 609.143,A -85,B 0,C 180,E1 29348.357,E2 29348.357} C_VEL
LIN {X 0,Y 632.89,Z 609.147,A -85,B 0,C 180,E1 29345.258,E2 29345.258} C_VEL
LIN {X 0,Y 632.89,Z 609.147,A -85,B 0,C 180,E1 29342.082,E2 29342.082} C_VEL
LIN {X 0,Y 632.891,Z 609.144,A -85,B 0,C 180,E1 29338.914,E2 29338.914} C_VEL
LIN {X 0,Y 632.888,Z 609.144,A -85,B 0,C 180,E1 29335.742,E2 29335.742} C_VEL
LIN {X 0,Y 632.896,Z 609.143,A -85,B 0,C 180,E1 29332.556,E2 29332.556} C_VEL
LIN {X 0,Y 632.89,Z 609.144,A -85,B 0,C 180,E1 29329.348,E2 29329.348} C_VEL
LIN {X 0,Y 632.895,Z 609.143,A -85,B 0,C 180,E1 29326.198,E2 29326.198} C_VEL
LIN {X 0,Y 632.89,Z 609.144,A -85,B 0,C 180,E1 29323.006,E2 29323.006} C_VEL
LIN {X 0,Y 632.892,Z 609.144,A -85,B 0,C 180,E1 29319.786,E2 29319.786} C_VEL
LIN {X 0,Y 632.89,Z 609.143,A -85,B 0,C 180,E1 29316.617,E2 29316.617} C_VEL
LIN {X 0,Y 632.889,Z 609.143,A -85,B 0,C 180,E1 29313.442,E2 29313.442} C_VEL
LIN {X 0,Y 632.891,Z 609.146,A -85,B 0,C 180,E1 29310.259,E2 29310.259} C_VEL
LIN {X 0,Y 632.891,Z 609.149,A -85,B 0,C 180,E1 29307.079,E2 29307.079} C_VEL
LIN {X 0,Y 632.886,Z 609.147,A -85,B 0,C 180,E1 29303.893,E2 29303.893} C_VEL
LIN {X 0,Y 632.894,Z 609.144,A -85,B 0,C 180,E1 29300.724,E2 29300.724} C_VEL
LIN {X 0,Y 632.891,Z 609.134,A -85,B 0,C 180,E1 29297.676,E2 29297.676} C_VEL
LIN {X 0,Y 632.892,Z 609.144,A -85,B 0,C 180,E1 29294.542,E2 29294.542} C_VEL
LIN {X 0,Y 632.895,Z 609.133,A -85,B 0,C 180,E1 29291.327,E2 29291.327} C_VEL
LIN {X 0,Y 632.89,Z 609.134,A -85,B 0,C 180,E1 29291.257,E2 29291.257} C_VEL
LIN {X 0,Y 631.871,Z 609.27,A -85,B 0,C 180,E1 29290.559,E2 29290.559} C_VEL
LIN {X 0,Y 625.46,Z 610.073,A -85,B 0,C 180,E1 29288.604,E2 29288.604} C_VEL
LIN {X 0,Y 624.948,Z 610.129,A -85,B 0,C 180,E1 29288.095,E2 29288.095} C_VEL
LIN {X 0,Y 624.953,Z 610.13,A -85,B 0,C 180,E1 29284.942,E2 29284.942} C_VEL
LIN {X 0,Y 624.945,Z 610.183,A -85,B 0,C 180,E1 29282.572,E2 29282.572} C_VEL
LIN {X 0,Y 633.076,Z 636.237,A -85,B 0,C 180,E1 29280.462,E2 29280.462} C_VEL
LIN {X 0,Y 632.487,Z 671.625,A -85,B 0,C 180,E1 29278.058,E2 29278.058} C_VEL
LIN {X 0,Y 631.415,Z 712.92,A -85,B 0,C 180,E1 29275.211,E2 29275.211} C_VEL
LIN {X 0,Y 630.182,Z 757.346,A -85,B 0,C 180,E1 29272.136,E2 29272.136} C_VEL
LIN {X 0,Y 629.033,Z 804.838,A -85,B 0,C 180,E1 29268.92,E2 29268.92} C_VEL
LIN {X 0,Y 628.541,Z 837.035,A -85,B 0,C 180,E1 29266.826,E2 29266.826} C_VEL
LIN {X 0,Y 629.358,Z 846.117,A -85,B 0,C 180,E1 29266.694,E2 29266.694} C_VEL
LIN {X 0,Y 628.274,Z 1006.384,A -85,B 0,C 180,E1 29264.818,E2 29264.818} C_VEL
LIN {X 0,Y 628.071,Z 1023.826,A -85,B 0,C 180,E1 29264.446,E2 29264.446} C_VEL
LIN {X 0,Y 627.723,Z 1040.405,A -85,B 0,C 180,E1 29263.916,E2 29263.916} C_VEL
LIN {X 0,Y 627.274,Z 1056.561,A -85,B 0,C 180,E1 29263.222,E2 29263.222} C_VEL
LIN {X 0,Y 626.771,Z 1071.683,A -85,B 0,C 180,E1 29262.389,E2 29262.389} C_VEL
LIN {X 0,Y 626.241,Z 1085.731,A -85,B 0,C 180,E1 29261.418,E2 29261.418} C_VEL
LIN {X 0,Y 625.719,Z 1098.711,A -85,B 0,C 180,E1 29260.309,E2 29260.309} C_VEL
LIN {X 0,Y 625.255,Z 1110.202,A -85,B 0,C 180,E1 29259.108,E2 29259.108} C_VEL
LIN {X 0,Y 624.869,Z 1120.286,A -85,B 0,C 180,E1 29257.816,E2 29257.816} C_VEL
LIN {X 0,Y 624.567,Z 1128.934,A -85,B 0,C 180,E1 29256.433,E2 29256.433} C_VEL
LIN {X 0,Y 624.357,Z 1136.135,A -85,B 0,C 180,E1 29254.96,E2 29254.96} C_VEL
LIN {X 0,Y 624.226,Z 1141.839,A -85,B 0,C 180,E1 29253.396,E2 29253.396} C_VEL
LIN {X 0,Y 624.15,Z 1145.739,A -85,B 0,C 180,E1 29251.835,E2 29251.835} C_VEL
LIN {X 0,Y 624.126,Z 1147.974,A -85,B 0,C 180,E1 29250.182,E2 29250.182} C_VEL
LIN {X 0,Y 624.111,Z 1148.411,A -85,B 0,C 180,E1 29248.53,E2 29248.53} C_VEL
LIN {X 0,Y 624.133,Z 1147.07,A -85,B 0,C 180,E1 29246.876,E2 29246.876} C_VEL
LIN {X 0,Y 624.183,Z 1144.065,A -85,B 0,C 180,E1 29245.313,E2 29245.313} C_VEL
LIN {X 0,Y 624.287,Z 1139.283,A -85,B 0,C 180,E1 29243.746,E2 29243.746} C_VEL
LIN {X 0,Y 624.457,Z 1132.61,A -85,B 0,C 180,E1 29242.176,E2 29242.176} C_VEL
LIN {X 0,Y 624.729,Z 1124.321,A -85,B 0,C 180,E1 29240.696,E2 29240.696} C_VEL
LIN {X 0,Y 625.09,Z 1114.393,A -85,B 0,C 180,E1 29239.306,E2 29239.306} C_VEL
LIN {X 0,Y 625.557,Z 1102.891,A -85,B 0,C 180,E1 29238.006,E2 29238.006} C_VEL
LIN {X 0,Y 626.075,Z 1090.191,A -85,B 0,C 180,E1 29236.844,E2 29236.844} C_VEL
LIN {X 0,Y 626.604,Z 1076.329,A -85,B 0,C 180,E1 29235.82,E2 29235.82} C_VEL
LIN {X 0,Y 627.121,Z 1061.464,A -85,B 0,C 180,E1 29234.935,E2 29234.935} C_VEL
LIN {X 0,Y 627.599,Z 1045.541,A -85,B 0,C 180,E1 29234.19,E2 29234.19} C_VEL
LIN {X 0,Y 627.978,Z 1028.723,A -85,B 0,C 180,E1 29233.603,E2 29233.603} C_VEL
LIN {X 0,Y 628.24,Z 1010.693,A -85,B 0,C 180,E1 29233.168,E2 29233.168} C_VEL
LIN {X 0,Y 628.374,Z 990.455,A -85,B 0,C 180,E1 29232.883,E2 29232.883} C_VEL
LIN {X 0,Y 629.154,Z 841.795,A -85,B 0,C 180,E1 29231.158,E2 29231.158} C_VEL
LIN {X 0,Y 628.484,Z 836.326,A -85,B 0,C 180,E1 29231.06,E2 29231.06} C_VEL
LIN {X 0,Y 629.458,Z 786.974,A -85,B 0,C 180,E1 29227.785,E2 29227.785} C_VEL
LIN {X 0,Y 630.691,Z 740.753,A -85,B 0,C 180,E1 29224.61,E2 29224.61} C_VEL
LIN {X 0,Y 631.946,Z 697.629,A -85,B 0,C 180,E1 29221.61,E2 29221.61} C_VEL
LIN {X 0,Y 632.975,Z 655.66,A -85,B 0,C 180,E1 29218.716,E2 29218.716} C_VEL
LIN {X 0,Y 633.245,Z 636.49,A -85,B 0,C 180,E1 29217.422,E2 29217.422} C_VEL
LIN {X 0,Y 625.703,Z 612.671,A -85,B 0,C 180,E1 29215.466,E2 29215.466} C_VEL
LIN {X 0,Y 624.943,Z 610.133,A -85,B 0,C 180,E1 29215.25,E2 29215.25} C_VEL
LIN {X 0,Y 624.935,Z 610.134,A -85,B 0,C 180,E1 29212.073,E2 29212.073} C_VEL
LIN {X 0,Y 624.95,Z 610.127,A -85,B 0,C 180,E1 29209.005,E2 29209.005} C_VEL
LIN {X 0,Y 624.936,Z 610.133,A -85,B 0,C 180,E1 29205.893,E2 29205.893} C_VEL
LIN {X 0,Y 624.937,Z 610.133,A -85,B 0,C 180,E1 29202.843,E2 29202.843} C_VEL
LIN {X 0,Y 624.952,Z 610.134,A -85,B 0,C 180,E1 29199.791,E2 29199.791} C_VEL
LIN {X 0,Y 624.941,Z 610.135,A -85,B 0,C 180,E1 29196.641,E2 29196.641} C_VEL
LIN {X 0,Y 624.984,Z 610.325,A -85,B 0,C 180,E1 29193.611,E2 29193.611} C_VEL
LIN {X 0,Y 627.037,Z 615.647,A -85,B 0,C 180,E1 29192.947,E2 29192.947} C_VEL
LIN {X 0,Y 638.063,Z 632.404,A -85,B 0,C 180,E1 29191.943,E2 29191.943} C_VEL
LIN {X 0,Y 643.99,Z 642.733,A -85,B 0,C 180,E1 29191.403,E2 29191.403} C_VEL
LIN {X 0,Y 639.965,Z 867.434,A -85,B 0,C 180,E1 29188.491,E2 29188.491} C_VEL
LIN {X 0,Y 638.749,Z 951.649,A -85,B 0,C 180,E1 29187.422,E2 29187.422} C_VEL
LIN {X 0,Y 638.015,Z 976.275,A -85,B 0,C 180,E1 29186.939,E2 29186.939} C_VEL
LIN {X 0,Y 637.108,Z 998.971,A -85,B 0,C 180,E1 29186.324,E2 29186.324} C_VEL
LIN {X 0,Y 636.084,Z 1020.1,A -85,B 0,C 180,E1 29185.59,E2 29185.59} C_VEL
LIN {X 0,Y 634.745,Z 1042.604,A -85,B 0,C 180,E1 29184.629,E2 29184.629} C_VEL
LIN {X 0,Y 633.504,Z 1061.927,A -85,B 0,C 180,E1 29183.635,E2 29183.635} C_VEL
LIN {X 0,Y 632.192,Z 1080.752,A -85,B 0,C 180,E1 29182.504,E2 29182.504} C_VEL
LIN {X 0,Y 630.605,Z 1102.034,A -85,B 0,C 180,E1 29180.999,E2 29180.999} C_VEL
LIN {X 0,Y 629.391,Z 1117.968,A -85,B 0,C 180,E1 29179.682,E2 29179.682} C_VEL
LIN {X 0,Y 628.32,Z 1132.088,A -85,B 0,C 180,E1 29178.366,E2 29178.366} C_VEL
LIN {X 0,Y 627.428,Z 1144.695,A -85,B 0,C 180,E1 29177.051,E2 29177.051} C_VEL
LIN {X 0,Y 626.617,Z 1156.737,A -85,B 0,C 180,E1 29175.645,E2 29175.645} C_VEL
LIN {X 0,Y 625.942,Z 1167.462,A -85,B 0,C 180,E1 29174.241,E2 29174.241} C_VEL
LIN {X 0,Y 625.334,Z 1178.195,A -85,B 0,C 180,E1 29172.654,E2 29172.654} C_VEL
LIN {X 0,Y 624.855,Z 1187.581,A -85,B 0,C 180,E1 29171.071,E2 29171.071} C_VEL
LIN {X 0,Y 624.521,Z 1195.752,A -85,B 0,C 180,E1 29169.492,E2 29169.492} C_VEL
LIN {X 0,Y 624.245,Z 1203.57,A -85,B 0,C 180,E1 29167.733,E2 29167.733} C_VEL
LIN {X 0,Y 624.059,Z 1211.037,A -85,B 0,C 180,E1 29165.701,E2 29165.701} C_VEL
LIN {X 0,Y 623.954,Z 1217.195,A -85,B 0,C 180,E1 29163.491,E2 29163.491} C_VEL
LIN {X 0,Y 623.917,Z 1221.084,A -85,B 0,C 180,E1 29161.561,E2 29161.561} C_VEL
LIN {X 0,Y 623.907,Z 1223.528,A -85,B 0,C 180,E1 29159.725,E2 29159.725} C_VEL
LIN {X 0,Y 623.91,Z 1224.714,A -85,B 0,C 180,E1 29157.979,E2 29157.979} C_VEL
LIN {X 0,Y 623.914,Z 1224.799,A -85,B 0,C 180,E1 29156.233,E2 29156.233} C_VEL
LIN {X 0,Y 623.911,Z 1223.804,A -85,B 0,C 180,E1 29154.482,E2 29154.482} C_VEL
LIN {X 0,Y 623.92,Z 1221.547,A -85,B 0,C 180,E1 29152.634,E2 29152.634} C_VEL
LIN {X 0,Y 623.954,Z 1217.825,A -85,B 0,C 180,E1 29150.685,E2 29150.685} C_VEL
LIN {X 0,Y 624.053,Z 1211.478,A -85,B 0,C 180,E1 29148.353,E2 29148.353} C_VEL
LIN {X 0,Y 624.227,Z 1204.384,A -85,B 0,C 180,E1 29146.381,E2 29146.381} C_VEL
LIN {X 0,Y 624.464,Z 1197.009,A -85,B 0,C 180,E1 29144.681,E2 29144.681} C_VEL
LIN {X 0,Y 624.807,Z 1188.829,A -85,B 0,C 180,E1 29143.067,E2 29143.067} C_VEL
LIN {X 0,Y 625.255,Z 1179.71,A -85,B 0,C 180,E1 29141.499,E2 29141.499} C_VEL
LIN {X 0,Y 625.807,Z 1169.579,A -85,B 0,C 180,E1 29139.966,E2 29139.966} C_VEL
LIN {X 0,Y 626.513,Z 1158.34,A -85,B 0,C 180,E1 29138.465,E2 29138.465} C_VEL
LIN {X 0,Y 627.33,Z 1146.102,A -85,B 0,C 180,E1 29137.014,E2 29137.014} C_VEL
LIN {X 0,Y 628.333,Z 1132.085,A -85,B 0,C 180,E1 29135.54,E2 29135.54} C_VEL
LIN {X 0,Y 629.711,Z 1113.659,A -85,B 0,C 180,E1 29133.856,E2 29133.856} C_VEL
LIN {X 0,Y 630.914,Z 1096.694,A -85,B 0,C 180,E1 29132.536,E2 29132.536} C_VEL
LIN {X 0,Y 632.011,Z 1080.858,A -85,B 0,C 180,E1 29131.459,E2 29131.459} C_VEL
LIN {X 0,Y 633.252,Z 1061.697,A -85,B 0,C 180,E1 29130.329,E2 29130.329} C_VEL
LIN {X 0,Y 634.479,Z 1039.506,A -85,B 0,C 180,E1 29129.244,E2 29129.244} C_VEL
LIN {X 0,Y 635.43,Z 1019.054,A -85,B 0,C 180,E1 29128.432,E2 29128.432} C_VEL
LIN {X 0,Y 636.233,Z 997.638,A -85,B 0,C 180,E1 29127.736,E2 29127.736} C_VEL
LIN {X 0,Y 636.824,Z 975.769,A -85,B 0,C 180,E1 29127.201,E2 29127.201} C_VEL
LIN {X 0,Y 637.267,Z 951.654,A -85,B 0,C 180,E1 29126.784,E2 29126.784} C_VEL
LIN {X 0,Y 638.628,Z 716.263,A -85,B 0,C 180,E1 29124.141,E2 29124.141} C_VEL
LIN {X 0,Y 639.131,Z 642.283,A -85,B 0,C 180,E1 29123.251,E2 29123.251} C_VEL
LIN {X 0,Y 637.442,Z 640.62,A -85,B 0,C 180,E1 29123.148,E2 29123.148} C_VEL
LIN {X 0,Y 637.919,Z 641.465,A -85,B 0,C 180,E1 29121.893,E2 29121.893} C_VEL
LIN {X 0,Y 639.039,Z 644.691,A -85,B 0,C 180,E1 29120.561,E2 29120.561} C_VEL
LIN {X 0,Y 639.205,Z 646.242,A -85,B 0,C 180,E1 29120.181,E2 29120.181} C_VEL
LIN {X 0,Y 634.701,Z 656.68,A -85,B 0,C 180,E1 29118.992,E2 29118.992} C_VEL
LIN {X 0,Y 631.256,Z 668.883,A -85,B 0,C 180,E1 29117.809,E2 29117.809} C_VEL
LIN {X 0,Y 628.666,Z 683.99,A -85,B 0,C 180,E1 29116.565,E2 29116.565} C_VEL
LIN {X 0,Y 626.753,Z 703.897,A -85,B 0,C 180,E1 29115.158,E2 29115.158} C_VEL
LIN {X 0,Y 625.384,Z 732.717,A -85,B 0,C 180,E1 29113.375,E2 29113.375} C_VEL
LIN {X 0,Y 625.055,Z 773.167,A -85,B 0,C 180,E1 29111.07,E2 29111.07} C_VEL
LIN {X 0,Y 626.774,Z 794.106,A -85,B 0,C 180,E1 29109.884,E2 29109.884} C_VEL
LIN {X 0,Y 630.057,Z 811.594,A -85,B 0,C 180,E1 29108.884,E2 29108.884} C_VEL
LIN {X 0,Y 634.963,Z 827.037,A -85,B 0,C 180,E1 29107.994,E2 29107.994} C_VEL
LIN {X 0,Y 641.686,Z 841.613,A -85,B 0,C 180,E1 29107.152,E2 29107.152} C_VEL
LIN {X 0,Y 649.788,Z 854.58,A -85,B 0,C 180,E1 29106.41,E2 29106.41} C_VEL
LIN {X 0,Y 659.201,Z 866.168,A -85,B 0,C 180,E1 29105.757,E2 29105.757} C_VEL
LIN {X 0,Y 670.275,Z 876.948,A -85,B 0,C 180,E1 29105.166,E2 29105.166} C_VEL
LIN {X 0,Y 682.102,Z 886.098,A -85,B 0,C 180,E1 29104.677,E2 29104.677} C_VEL
LIN {X 0,Y 693.513,Z 893.154,A -85,B 0,C 180,E1 29104.295,E2 29104.295} C_VEL
LIN {X 0,Y 697.6,Z 894.917,A -85,B 0,C 180,E1 29104.099,E2 29104.099} C_VEL
LIN {X 0,Y 690.512,Z 902.813,A -85,B 0,C 180,E1 29103.78,E2 29103.78} C_VEL
LIN {X 0,Y 673.568,Z 915.971,A -85,B 0,C 180,E1 29103.113,E2 29103.113} C_VEL
LIN {X 0,Y 661.944,Z 926.809,A -85,B 0,C 180,E1 29102.531,E2 29102.531} C_VEL
LIN {X 0,Y 653.517,Z 936.932,A -85,B 0,C 180,E1 29101.965,E2 29101.965} C_VEL
LIN {X 0,Y 642.161,Z 955.465,A -85,B 0,C 180,E1 29100.913,E2 29100.913} C_VEL
LIN {X 0,Y 640.236,Z 959.892,A -85,B 0,C 180,E1 29100.688,E2 29100.688} C_VEL
LIN {X 0,Y 637.581,Z 970.759,A -85,B 0,C 180,E1 29100.64,E2 29100.64} C_VEL
LIN {X 0,Y 637.128,Z 984.098,A -85,B 0,C 180,E1 29100.501,E2 29100.501} C_VEL
LIN {X 0,Y 636.7,Z 1013.869,A -85,B 0,C 180,E1 29100.106,E2 29100.106} C_VEL
LIN {X 0,Y 636.001,Z 1040.616,A -85,B 0,C 180,E1 29099.582,E2 29099.582} C_VEL
LIN {X 0,Y 635.176,Z 1065.857,A -85,B 0,C 180,E1 29098.925,E2 29098.925} C_VEL
LIN {X 0,Y 634.345,Z 1089.238,A -85,B 0,C 180,E1 29098.165,E2 29098.165} C_VEL
LIN {X 0,Y 633.384,Z 1112.473,A -85,B 0,C 180,E1 29097.247,E2 29097.247} C_VEL
LIN {X 0,Y 632.355,Z 1135.011,A -85,B 0,C 180,E1 29096.179,E2 29096.179} C_VEL
LIN {X 0,Y 631.248,Z 1156.484,A -85,B 0,C 180,E1 29094.973,E2 29094.973} C_VEL
LIN {X 0,Y 630.196,Z 1175.409,A -85,B 0,C 180,E1 29093.724,E2 29093.724} C_VEL
LIN {X 0,Y 629.086,Z 1191.942,A -85,B 0,C 180,E1 29092.376,E2 29092.376} C_VEL
LIN {X 0,Y 627.965,Z 1207.199,A -85,B 0,C 180,E1 29090.897,E2 29090.897} C_VEL
LIN {X 0,Y 627.047,Z 1220.249,A -85,B 0,C 180,E1 29089.468,E2 29089.468} C_VEL
LIN {X 0,Y 626.286,Z 1231.826,A -85,B 0,C 180,E1 29088.044,E2 29088.044} C_VEL
LIN {X 0,Y 625.674,Z 1242.108,A -85,B 0,C 180,E1 29086.623,E2 29086.623} C_VEL
LIN {X 0,Y 625.135,Z 1251.815,A -85,B 0,C 180,E1 29085.114,E2 29085.114} C_VEL
LIN {X 0,Y 624.721,Z 1260.839,A -85,B 0,C 180,E1 29083.515,E2 29083.515} C_VEL
LIN {X 0,Y 624.377,Z 1269.935,A -85,B 0,C 180,E1 29081.642,E2 29081.642} C_VEL
LIN {X 0,Y 624.118,Z 1278.783,A -85,B 0,C 180,E1 29079.406,E2 29079.406} C_VEL
LIN {X 0,Y 623.995,Z 1284.807,A -85,B 0,C 180,E1 29077.459,E2 29077.459} C_VEL
LIN {X 0,Y 623.924,Z 1289.031,A -85,B 0,C 180,E1 29075.703,E2 29075.703} C_VEL
LIN {X 0,Y 623.902,Z 1292.37,A -85,B 0,C 180,E1 29073.769,E2 29073.769} C_VEL
LIN {X 0,Y 623.893,Z 1294.558,A -85,B 0,C 180,E1 29071.562,E2 29071.562} C_VEL
LIN {X 0,Y 623.893,Z 1294.862,A -85,B 0,C 180,E1 29069.45,E2 29069.45} C_VEL
LIN {X 0,Y 623.899,Z 1293.887,A -85,B 0,C 180,E1 29067.613,E2 29067.613} C_VEL
LIN {X 0,Y 623.914,Z 1291.692,A -85,B 0,C 180,E1 29065.774,E2 29065.774} C_VEL
LIN {X 0,Y 623.942,Z 1288.255,A -85,B 0,C 180,E1 29063.93,E2 29063.93} C_VEL
LIN {X 0,Y 624.04,Z 1282.485,A -85,B 0,C 180,E1 29061.71,E2 29061.71} C_VEL
LIN {X 0,Y 624.199,Z 1275.34,A -85,B 0,C 180,E1 29059.666,E2 29059.666} C_VEL
LIN {X 0,Y 624.45,Z 1267.795,A -85,B 0,C 180,E1 29057.893,E2 29057.893} C_VEL
LIN {X 0,Y 624.785,Z 1259.352,A -85,B 0,C 180,E1 29056.206,E2 29056.206} C_VEL
LIN {X 0,Y 625.232,Z 1250.111,A -85,B 0,C 180,E1 29054.607,E2 29054.607} C_VEL
LIN {X 0,Y 625.906,Z 1238.204,A -85,B 0,C 180,E1 29052.807,E2 29052.807} C_VEL
LIN {X 0,Y 626.831,Z 1223.546,A -85,B 0,C 180,E1 29050.914,E2 29050.914} C_VEL
LIN {X 0,Y 627.763,Z 1209.966,A -85,B 0,C 180,E1 29049.392,E2 29049.392} C_VEL
LIN {X 0,Y 628.741,Z 1196.561,A -85,B 0,C 180,E1 29048.056,E2 29048.056} C_VEL
LIN {X 0,Y 629.55,Z 1185.273,A -85,B 0,C 180,E1 29047.052,E2 29047.052} C_VEL
LIN {X 0,Y 630.769,Z 1167.359,A -85,B 0,C 180,E1 29045.662,E2 29045.662} C_VEL
LIN {X 0,Y 632.186,Z 1146.188,A -85,B 0,C 180,E1 29044.252,E2 29044.252} C_VEL
LIN {X 0,Y 633.595,Z 1124.505,A -85,B 0,C 180,E1 29043.02,E2 29043.02} C_VEL
LIN {X 0,Y 634.977,Z 1102.201,A -85,B 0,C 180,E1 29041.951,E2 29041.951} C_VEL
LIN {X 0,Y 636.308,Z 1079.173,A -85,B 0,C 180,E1 29041.027,E2 29041.027} C_VEL
LIN {X 0,Y 637.548,Z 1056.154,A -85,B 0,C 180,E1 29040.287,E2 29040.287} C_VEL
LIN {X 0,Y 638.625,Z 1033.369,A -85,B 0,C 180,E1 29039.704,E2 29039.704} C_VEL
LIN {X 0,Y 639.496,Z 1010.209,A -85,B 0,C 180,E1 29039.279,E2 29039.279} C_VEL
LIN {X 0,Y 640.51,Z 970.705,A -85,B 0,C 180,E1 29038.772,E2 29038.772} C_VEL
LIN {X 0,Y 640.806,Z 968.375,A -85,B 0,C 180,E1 29038.749,E2 29038.749} C_VEL
LIN {X 0,Y 646.348,Z 956.909,A -85,B 0,C 180,E1 29038.136,E2 29038.136} C_VEL
LIN {X 0,Y 656.646,Z 939.924,A -85,B 0,C 180,E1 29037.332,E2 29037.332} C_VEL
LIN {X 0,Y 665.37,Z 928.682,A -85,B 0,C 180,E1 29036.892,E2 29036.892} C_VEL
LIN {X 0,Y 677.559,Z 915.731,A -85,B 0,C 180,E1 29036.49,E2 29036.49} C_VEL
LIN {X 0,Y 691.886,Z 902.099,A -85,B 0,C 180,E1 29036.146,E2 29036.146} C_VEL
LIN {X 0,Y 697.562,Z 894.863,A -85,B 0,C 180,E1 29035.885,E2 29035.885} C_VEL
LIN {X 0,Y 685.528,Z 890.699,A -85,B 0,C 180,E1 29035.057,E2 29035.057} C_VEL
LIN {X 0,Y 674.723,Z 885.244,A -85,B 0,C 180,E1 29034.156,E2 29034.156} C_VEL
LIN {X 0,Y 664.813,Z 878.19,A -85,B 0,C 180,E1 29033.144,E2 29033.144} C_VEL
LIN {X 0,Y 656.551,Z 869.894,A -85,B 0,C 180,E1 29032.082,E2 29032.082} C_VEL
LIN {X 0,Y 649.932,Z 860.409,A -85,B 0,C 180,E1 29030.98,E2 29030.98} C_VEL
LIN {X 0,Y 644.572,Z 848.821,A -85,B 0,C 180,E1 29029.749,E2 29029.749} C_VEL
LIN {X 0,Y 641.157,Z 836.317,A -85,B 0,C 180,E1 29028.534,E2 29028.534} C_VEL
LIN {X 0,Y 639.493,Z 821.831,A -85,B 0,C 180,E1 29027.238,E2 29027.238} C_VEL
LIN {X 0,Y 639.629,Z 803.474,A -85,B 0,C 180,E1 29025.722,E2 29025.722} C_VEL
LIN {X 0,Y 641.893,Z 765.571,A -85,B 0,C 180,E1 29022.657,E2 29022.657} C_VEL
LIN {X 0,Y 644.068,Z 729.856,A -85,B 0,C 180,E1 29019.7,E2 29019.7} C_VEL
LIN {X 0,Y 646.142,Z 695.681,A -85,B 0,C 180,E1 29016.789,E2 29016.789} C_VEL
LIN {X 0,Y 648.083,Z 663.39,A -85,B 0,C 180,E1 29013.953,E2 29013.953} C_VEL
LIN {X 0,Y 639.677,Z 643.598,A -85,B 0,C 180,E1 29011.241,E2 29011.241} C_VEL
LIN {X 0,Y 631.867,Z 625.866,A -85,B 0,C 180,E1 29008.652,E2 29008.652} C_VEL
LIN {X 0,Y 627.756,Z 617.052,A -85,B 0,C 180,E1 29007.284,E2 29007.284} C_VEL
LIN {X 0,Y 626.263,Z 613.639,A -85,B 0,C 180,E1 29006.759,E2 29006.759} C_VEL
LIN {X 0,Y 624.955,Z 610.132,A -85,B 0,C 180,E1 29006.205,E2 29006.205} C_VEL
LIN {X 0,Y 624.94,Z 610.137,A -85,B 0,C 180,E1 29003.079,E2 29003.079} C_VEL
LIN {X 0,Y 624.952,Z 610.136,A -85,B 0,C 180,E1 28999.925,E2 28999.925} C_VEL
LIN {X 0,Y 624.936,Z 610.133,A -85,B 0,C 180,E1 28996.834,E2 28996.834} C_VEL
LIN {X 0,Y 624.946,Z 610.136,A -85,B 0,C 180,E1 28993.697,E2 28993.697} C_VEL
LIN {X 0,Y 624.938,Z 610.13,A -85,B 0,C 180,E1 28990.603,E2 28990.603} C_VEL
LIN {X 0,Y 624.939,Z 610.134,A -85,B 0,C 180,E1 28987.446,E2 28987.446} C_VEL
LIN {X 0,Y 624.935,Z 610.135,A -85,B 0,C 180,E1 28984.313,E2 28984.313} C_VEL
LIN {X 0,Y 624.935,Z 610.131,A -85,B 0,C 180,E1 28981.192,E2 28981.192} C_VEL
LIN {X 0,Y 624.939,Z 610.131,A -85,B 0,C 180,E1 28978.166,E2 28978.166} C_VEL
LIN {X 0,Y 624.939,Z 610.133,A -85,B 0,C 180,E1 28975.043,E2 28975.043} C_VEL
LIN {X 0,Y 624.939,Z 610.134,A -85,B 0,C 180,E1 28971.906,E2 28971.906} C_VEL
LIN {X 0,Y 624.939,Z 610.134,A -85,B 0,C 180,E1 28968.74,E2 28968.74} C_VEL
LIN {X 0,Y 624.938,Z 610.135,A -85,B 0,C 180,E1 28965.641,E2 28965.641} C_VEL
LIN {X 0,Y 624.938,Z 610.135,A -85,B 0,C 180,E1 28962.469,E2 28962.469} C_VEL
LIN {X 0,Y 624.938,Z 610.134,A -85,B 0,C 180,E1 28959.383,E2 28959.383} C_VEL
LIN {X 0,Y 624.939,Z 610.133,A -85,B 0,C 180,E1 28956.322,E2 28956.322} C_VEL
LIN {X 0,Y 624.943,Z 610.13,A -85,B 0,C 180,E1 28953.221,E2 28953.221} C_VEL
LIN {X 0,Y 624.94,Z 610.133,A -85,B 0,C 180,E1 28950.053,E2 28950.053} C_VEL
LIN {X 0,Y 624.946,Z 610.136,A -85,B 0,C 180,E1 28946.935,E2 28946.935} C_VEL
LIN {X 0,Y 624.938,Z 610.138,A -85,B 0,C 180,E1 28943.741,E2 28943.741} C_VEL
LIN {X 0,Y 624.951,Z 610.135,A -85,B 0,C 180,E1 28940.601,E2 28940.601} C_VEL
LIN {X 0,Y 624.944,Z 610.12,A -85,B 0,C 180,E1 28937.523,E2 28937.523} C_VEL
LIN {X 0,Y 624.954,Z 610.136,A -85,B 0,C 180,E1 28934.342,E2 28934.342} C_VEL
LIN {X 0,Y 624.95,Z 610.122,A -85,B 0,C 180,E1 28931.235,E2 28931.235} C_VEL
LIN {X 0,Y 624.948,Z 610.129,A -85,B 0,C 180,E1 28928.095,E2 28928.095} C_VEL
LIN {X 0,Y 623.984,Z 610.246,A -85,B 0,C 180,E1 28927.389,E2 28927.389} C_VEL
LIN {X 0,Y 617.56,Z 611.06,A -85,B 0,C 180,E1 28925.409,E2 28925.409} C_VEL
LIN {X 0,Y 617.012,Z 611.118,A -85,B 0,C 180,E1 28924.894,E2 28924.894} C_VEL
LIN {X 0,Y 617.009,Z 611.206,A -85,B 0,C 180,E1 28922.897,E2 28922.897} C_VEL
LIN {X 0,Y 625.622,Z 638.614,A -85,B 0,C 180,E1 28920.651,E2 28920.651} C_VEL
LIN {X 0,Y 625.043,Z 673.573,A -85,B 0,C 180,E1 28918.261,E2 28918.261} C_VEL
LIN {X 0,Y 623.874,Z 715.926,A -85,B 0,C 180,E1 28915.32,E2 28915.32} C_VEL
LIN {X 0,Y 622.569,Z 761.189,A -85,B 0,C 180,E1 28912.173,E2 28912.173} C_VEL
LIN {X 0,Y 621.394,Z 807.945,A -85,B 0,C 180,E1 28908.996,E2 28908.996} C_VEL
LIN {X 0,Y 620.95,Z 837.902,A -85,B 0,C 180,E1 28907.05,E2 28907.05} C_VEL
LIN {X 0,Y 621.759,Z 846.908,A -85,B 0,C 180,E1 28906.917,E2 28906.917} C_VEL
LIN {X 0,Y 620.607,Z 1007.331,A -85,B 0,C 180,E1 28905.017,E2 28905.017} C_VEL
LIN {X 0,Y 620.401,Z 1024.755,A -85,B 0,C 180,E1 28904.641,E2 28904.641} C_VEL
LIN {X 0,Y 620.033,Z 1041.651,A -85,B 0,C 180,E1 28904.092,E2 28904.092} C_VEL
LIN {X 0,Y 619.566,Z 1057.751,A -85,B 0,C 180,E1 28903.389,E2 28903.389} C_VEL
LIN {X 0,Y 619.037,Z 1072.832,A -85,B 0,C 180,E1 28902.546,E2 28902.546} C_VEL
LIN {X 0,Y 618.471,Z 1086.938,A -85,B 0,C 180,E1 28901.555,E2 28901.555} C_VEL
LIN {X 0,Y 617.923,Z 1099.791,A -85,B 0,C 180,E1 28900.44,E2 28900.44} C_VEL
LIN {X 0,Y 617.426,Z 1111.262,A -85,B 0,C 180,E1 28899.224,E2 28899.224} C_VEL
LIN {X 0,Y 617.01,Z 1121.328,A -85,B 0,C 180,E1 28897.916,E2 28897.916} C_VEL
LIN {X 0,Y 616.68,Z 1129.953,A -85,B 0,C 180,E1 28896.516,E2 28896.516} C_VEL
LIN {X 0,Y 616.448,Z 1137.14,A -85,B 0,C 180,E1 28895.024,E2 28895.024} C_VEL
LIN {X 0,Y 616.3,Z 1142.831,A -85,B 0,C 180,E1 28893.44,E2 28893.44} C_VEL
LIN {X 0,Y 616.214,Z 1146.718,A -85,B 0,C 180,E1 28891.858,E2 28891.858} C_VEL
LIN {X 0,Y 616.184,Z 1148.935,A -85,B 0,C 180,E1 28890.185,E2 28890.185} C_VEL
LIN {X 0,Y 616.168,Z 1149.36,A -85,B 0,C 180,E1 28888.511,E2 28888.511} C_VEL
LIN {X 0,Y 616.194,Z 1148.008,A -85,B 0,C 180,E1 28886.836,E2 28886.836} C_VEL
LIN {X 0,Y 616.253,Z 1144.983,A -85,B 0,C 180,E1 28885.252,E2 28885.252} C_VEL
LIN {X 0,Y 616.371,Z 1140.187,A -85,B 0,C 180,E1 28883.666,E2 28883.666} C_VEL
LIN {X 0,Y 616.564,Z 1133.499,A -85,B 0,C 180,E1 28882.076,E2 28882.076} C_VEL
LIN {X 0,Y 616.843,Z 1125.781,A -85,B 0,C 180,E1 28880.67,E2 28880.67} C_VEL
LIN {X 0,Y 617.228,Z 1115.977,A -85,B 0,C 180,E1 28879.262,E2 28879.262} C_VEL
LIN {X 0,Y 617.72,Z 1104.6,A -85,B 0,C 180,E1 28877.946,E2 28877.946} C_VEL
LIN {X 0,Y 618.242,Z 1092.576,A -85,B 0,C 180,E1 28876.812,E2 28876.812} C_VEL
LIN {X 0,Y 618.798,Z 1079.183,A -85,B 0,C 180,E1 28875.781,E2 28875.781} C_VEL
LIN {X 0,Y 619.318,Z 1065.033,A -85,B 0,C 180,E1 28874.901,E2 28874.901} C_VEL
LIN {X 0,Y 619.82,Z 1049.412,A -85,B 0,C 180,E1 28874.13,E2 28874.13} C_VEL
LIN {X 0,Y 620.237,Z 1033.136,A -85,B 0,C 180,E1 28873.516,E2 28873.516} C_VEL
LIN {X 0,Y 620.532,Z 1016.068,A -85,B 0,C 180,E1 28873.057,E2 28873.057} C_VEL
LIN {X 0,Y 620.676,Z 997.658,A -85,B 0,C 180,E1 28872.753,E2 28872.753} C_VEL
LIN {X 0,Y 621.582,Z 842.666,A -85,B 0,C 180,E1 28870.932,E2 28870.932} C_VEL
LIN {X 0,Y 620.908,Z 837.01,A -85,B 0,C 180,E1 28870.82,E2 28870.82} C_VEL
LIN {X 0,Y 621.904,Z 787.871,A -85,B 0,C 180,E1 28867.551,E2 28867.551} C_VEL
LIN {X 0,Y 623.214,Z 741.258,A -85,B 0,C 180,E1 28864.329,E2 28864.329} C_VEL
LIN {X 0,Y 624.528,Z 697.88,A -85,B 0,C 180,E1 28861.293,E2 28861.293} C_VEL
LIN {X 0,Y 625.579,Z 657.402,A -85,B 0,C 180,E1 28858.488,E2 28858.488} C_VEL
LIN {X 0,Y 625.707,Z 638.538,A -85,B 0,C 180,E1 28857.198,E2 28857.198} C_VEL
LIN {X 0,Y 618.52,Z 615.952,A -85,B 0,C 180,E1 28855.316,E2 28855.316} C_VEL
LIN {X 0,Y 617.017,Z 611.127,A -85,B 0,C 180,E1 28854.922,E2 28854.922} C_VEL
LIN {X 0,Y 617.011,Z 611.124,A -85,B 0,C 180,E1 28851.634,E2 28851.634} C_VEL
LIN {X 0,Y 617.015,Z 611.12,A -85,B 0,C 180,E1 28848.337,E2 28848.337} C_VEL
LIN {X 0,Y 617.005,Z 611.122,A -85,B 0,C 180,E1 28845.043,E2 28845.043} C_VEL
LIN {X 0,Y 617.01,Z 611.121,A -85,B 0,C 180,E1 28841.887,E2 28841.887} C_VEL
LIN {X 0,Y 617.001,Z 611.122,A -85,B 0,C 180,E1 28838.722,E2 28838.722} C_VEL
LIN {X 0,Y 617.016,Z 611.122,A -85,B 0,C 180,E1 28835.559,E2 28835.559} C_VEL
LIN {X 0,Y 617.001,Z 611.146,A -85,B 0,C 180,E1 28834.259,E2 28834.259} C_VEL
LIN {X 0,Y 618.379,Z 614.695,A -85,B 0,C 180,E1 28833.786,E2 28833.786} C_VEL
LIN {X 0,Y 619.518,Z 617.566,A -85,B 0,C 180,E1 28833.443,E2 28833.443} C_VEL
LIN {X 0,Y 632.5,Z 637.072,A -85,B 0,C 180,E1 28832.246,E2 28832.246} C_VEL
LIN {X 0,Y 637.45,Z 645.824,A -85,B 0,C 180,E1 28831.784,E2 28831.784} C_VEL
LIN {X 0,Y 632.975,Z 872.469,A -85,B 0,C 180,E1 28828.793,E2 28828.793} C_VEL
LIN {X 0,Y 631.668,Z 953.504,A -85,B 0,C 180,E1 28827.738,E2 28827.738} C_VEL
LIN {X 0,Y 630.903,Z 977.245,A -85,B 0,C 180,E1 28827.26,E2 28827.26} C_VEL
LIN {X 0,Y 629.969,Z 999.846,A -85,B 0,C 180,E1 28826.64,E2 28826.64} C_VEL
LIN {X 0,Y 628.848,Z 1021.533,A -85,B 0,C 180,E1 28825.874,E2 28825.874} C_VEL
LIN {X 0,Y 627.483,Z 1043.212,A -85,B 0,C 180,E1 28824.933,E2 28824.933} C_VEL
LIN {X 0,Y 626.178,Z 1062.575,A -85,B 0,C 180,E1 28823.928,E2 28823.928} C_VEL
LIN {X 0,Y 624.734,Z 1082.094,A -85,B 0,C 180,E1 28822.738,E2 28822.738} C_VEL
LIN {X 0,Y 623.056,Z 1103.219,A -85,B 0,C 180,E1 28821.216,E2 28821.216} C_VEL
LIN {X 0,Y 621.78,Z 1119.1,A -85,B 0,C 180,E1 28819.884,E2 28819.884} C_VEL
LIN {X 0,Y 620.599,Z 1133.557,A -85,B 0,C 180,E1 28818.506,E2 28818.506} C_VEL
LIN {X 0,Y 619.639,Z 1145.923,A -85,B 0,C 180,E1 28817.176,E2 28817.176} C_VEL
LIN {X 0,Y 618.776,Z 1157.811,A -85,B 0,C 180,E1 28815.752,E2 28815.752} C_VEL
LIN {X 0,Y 618.033,Z 1168.779,A -85,B 0,C 180,E1 28814.279,E2 28814.279} C_VEL
LIN {X 0,Y 617.414,Z 1179.037,A -85,B 0,C 180,E1 28812.724,E2 28812.724} C_VEL
LIN {X 0,Y 616.909,Z 1188.321,A -85,B 0,C 180,E1 28811.121,E2 28811.121} C_VEL
LIN {X 0,Y 616.503,Z 1197.743,A -85,B 0,C 180,E1 28809.24,E2 28809.24} C_VEL
LIN {X 0,Y 616.175,Z 1207.309,A -85,B 0,C 180,E1 28806.897,E2 28806.897} C_VEL
LIN {X 0,Y 616.03,Z 1213.358,A -85,B 0,C 180,E1 28805.028,E2 28805.028} C_VEL
LIN {X 0,Y 615.954,Z 1217.889,A -85,B 0,C 180,E1 28803.257,E2 28803.257} C_VEL
LIN {X 0,Y 615.918,Z 1221.142,A -85,B 0,C 180,E1 28801.581,E2 28801.581} C_VEL
LIN {X 0,Y 615.907,Z 1223.472,A -85,B 0,C 180,E1 28799.814,E2 28799.814} C_VEL
LIN {X 0,Y 615.912,Z 1224.691,A -85,B 0,C 180,E1 28798.046,E2 28798.046} C_VEL
LIN {X 0,Y 615.914,Z 1224.81,A -85,B 0,C 180,E1 28796.277,E2 28796.277} C_VEL
LIN {X 0,Y 615.912,Z 1223.846,A -85,B 0,C 180,E1 28794.504,E2 28794.504} C_VEL
LIN {X 0,Y 615.921,Z 1221.62,A -85,B 0,C 180,E1 28792.632,E2 28792.632} C_VEL
LIN {X 0,Y 615.951,Z 1218.326,A -85,B 0,C 180,E1 28790.846,E2 28790.846} C_VEL
LIN {X 0,Y 616.018,Z 1213.591,A -85,B 0,C 180,E1 28788.958,E2 28788.958} C_VEL
LIN {X 0,Y 616.209,Z 1206.126,A -85,B 0,C 180,E1 28786.678,E2 28786.678} C_VEL
LIN {X 0,Y 616.49,Z 1197.708,A -85,B 0,C 180,E1 28784.67,E2 28784.67} C_VEL
LIN {X 0,Y 616.877,Z 1189.12,A -85,B 0,C 180,E1 28782.939,E2 28782.939} C_VEL
LIN {X 0,Y 617.359,Z 1180.034,A -85,B 0,C 180,E1 28781.35,E2 28781.35} C_VEL
LIN {X 0,Y 617.934,Z 1170.229,A -85,B 0,C 180,E1 28779.839,E2 28779.839} C_VEL
LIN {X 0,Y 618.655,Z 1159.525,A -85,B 0,C 180,E1 28778.377,E2 28778.377} C_VEL
LIN {X 0,Y 619.458,Z 1148.292,A -85,B 0,C 180,E1 28777.007,E2 28777.007} C_VEL
LIN {X 0,Y 620.421,Z 1135.725,A -85,B 0,C 180,E1 28775.633,E2 28775.633} C_VEL
LIN {X 0,Y 621.578,Z 1120.915,A -85,B 0,C 180,E1 28774.206,E2 28774.206} C_VEL
LIN {X 0,Y 622.997,Z 1102.535,A -85,B 0,C 180,E1 28772.676,E2 28772.676} C_VEL
LIN {X 0,Y 624.318,Z 1083.838,A -85,B 0,C 180,E1 28771.363,E2 28771.363} C_VEL
LIN {X 0,Y 625.633,Z 1064.51,A -85,B 0,C 180,E1 28770.195,E2 28770.195} C_VEL
LIN {X 0,Y 626.71,Z 1045.499,A -85,B 0,C 180,E1 28769.235,E2 28769.235} C_VEL
LIN {X 0,Y 627.8,Z 1023.668,A -85,B 0,C 180,E1 28768.319,E2 28768.319} C_VEL
LIN {X 0,Y 628.579,Z 1004.258,A -85,B 0,C 180,E1 28767.661,E2 28767.661} C_VEL
LIN {X 0,Y 629.242,Z 980.891,A -85,B 0,C 180,E1 28767.046,E2 28767.046} C_VEL
LIN {X 0,Y 629.688,Z 958.342,A -85,B 0,C 180,E1 28766.618,E2 28766.618} C_VEL
LIN {X 0,Y 630.069,Z 901.468,A -85,B 0,C 180,E1 28765.968,E2 28765.968} C_VEL
LIN {X 0,Y 631.201,Z 725.752,A -85,B 0,C 180,E1 28763.969,E2 28763.969} C_VEL
LIN {X 0,Y 631.904,Z 646.407,A -85,B 0,C 180,E1 28762.987,E2 28762.987} C_VEL
LIN {X 0,Y 631.132,Z 645.566,A -85,B 0,C 180,E1 28762.928,E2 28762.928} C_VEL
LIN {X 0,Y 631.694,Z 646.726,A -85,B 0,C 180,E1 28761.731,E2 28761.731} C_VEL
LIN {X 0,Y 632.711,Z 650.091,A -85,B 0,C 180,E1 28760.463,E2 28760.463} C_VEL
LIN {X 0,Y 627.912,Z 660.411,A -85,B 0,C 180,E1 28759.24,E2 28759.24} C_VEL
LIN {X 0,Y 624.179,Z 672.557,A -85,B 0,C 180,E1 28758.014,E2 28758.014} C_VEL
LIN {X 0,Y 621.325,Z 687.599,A -85,B 0,C 180,E1 28756.72,E2 28756.72} C_VEL
LIN {X 0,Y 619.282,Z 706.248,A -85,B 0,C 180,E1 28755.342,E2 28755.342} C_VEL
LIN {X 0,Y 617.743,Z 733.296,A -85,B 0,C 180,E1 28753.594,E2 28753.594} C_VEL
LIN {X 0,Y 617.146,Z 771.964,A -85,B 0,C 180,E1 28751.312,E2 28751.312} C_VEL
LIN {X 0,Y 618.662,Z 793.475,A -85,B 0,C 180,E1 28750.061,E2 28750.061} C_VEL
LIN {X 0,Y 621.926,Z 812.022,A -85,B 0,C 180,E1 28748.975,E2 28748.975} C_VEL
LIN {X 0,Y 626.655,Z 827.625,A -85,B 0,C 180,E1 28748.054,E2 28748.054} C_VEL
LIN {X 0,Y 633.485,Z 842.99,A -85,B 0,C 180,E1 28747.147,E2 28747.147} C_VEL
LIN {X 0,Y 641.793,Z 856.687,A -85,B 0,C 180,E1 28746.344,E2 28746.344} C_VEL
LIN {X 0,Y 651.066,Z 868.464,A -85,B 0,C 180,E1 28745.666,E2 28745.666} C_VEL
LIN {X 0,Y 661.979,Z 879.493,A -85,B 0,C 180,E1 28745.048,E2 28745.048} C_VEL
LIN {X 0,Y 674.534,Z 889.585,A -85,B 0,C 180,E1 28744.494,E2 28744.494} C_VEL
LIN {X 0,Y 685.917,Z 897.231,A -85,B 0,C 180,E1 28744.101,E2 28744.101} C_VEL
LIN {X 0,Y 665.506,Z 913.197,A -85,B 0,C 180,E1 28743.258,E2 28743.258} C_VEL
LIN {X 0,Y 654.079,Z 924.263,A -85,B 0,C 180,E1 28742.659,E2 28742.659} C_VEL
LIN {X 0,Y 645.759,Z 934.69,A -85,B 0,C 180,E1 28742.081,E2 28742.081} C_VEL
LIN {X 0,Y 634.793,Z 952.787,A -85,B 0,C 180,E1 28741.056,E2 28741.056} C_VEL
LIN {X 0,Y 633.677,Z 955.321,A -85,B 0,C 180,E1 28740.942,E2 28740.942} C_VEL
LIN {X 0,Y 630.214,Z 968.967,A -85,B 0,C 180,E1 28740.885,E2 28740.885} C_VEL
LIN {X 0,Y 629.571,Z 978.954,A -85,B 0,C 180,E1 28740.788,E2 28740.788} C_VEL
LIN {X 0,Y 629.118,Z 1009.554,A -85,B 0,C 180,E1 28740.376,E2 28740.376} C_VEL
LIN {X 0,Y 628.327,Z 1036.966,A -85,B 0,C 180,E1 28739.838,E2 28739.838} C_VEL
LIN {X 0,Y 627.435,Z 1063.054,A -85,B 0,C 180,E1 28739.155,E2 28739.155} C_VEL
LIN {X 0,Y 626.586,Z 1086.311,A -85,B 0,C 180,E1 28738.395,E2 28738.395} C_VEL
LIN {X 0,Y 625.586,Z 1109.763,A -85,B 0,C 180,E1 28737.469,E2 28737.469} C_VEL
LIN {X 0,Y 624.56,Z 1131.868,A -85,B 0,C 180,E1 28736.428,E2 28736.428} C_VEL
LIN {X 0,Y 623.453,Z 1153.266,A -85,B 0,C 180,E1 28735.238,E2 28735.238} C_VEL
LIN {X 0,Y 622.258,Z 1174.767,A -85,B 0,C 180,E1 28733.83,E2 28733.83} C_VEL
LIN {X 0,Y 621.126,Z 1192.776,A -85,B 0,C 180,E1 28732.429,E2 28732.429} C_VEL
LIN {X 0,Y 620.321,Z 1205.867,A -85,B 0,C 180,E1 28731.266,E2 28731.266} C_VEL
LIN {X 0,Y 619.507,Z 1217.799,A -85,B 0,C 180,E1 28730.01,E2 28730.01} C_VEL
LIN {X 0,Y 618.597,Z 1230.369,A -85,B 0,C 180,E1 28728.471,E2 28728.471} C_VEL
LIN {X 0,Y 617.868,Z 1241.46,A -85,B 0,C 180,E1 28726.936,E2 28726.936} C_VEL
LIN {X 0,Y 617.287,Z 1251.242,A -85,B 0,C 180,E1 28725.407,E2 28725.407} C_VEL
LIN {X 0,Y 616.818,Z 1260.336,A -85,B 0,C 180,E1 28723.787,E2 28723.787} C_VEL
LIN {X 0,Y 616.468,Z 1268.637,A -85,B 0,C 180,E1 28722.079,E2 28722.079} C_VEL
LIN {X 0,Y 616.193,Z 1276.411,A -85,B 0,C 180,E1 28720.189,E2 28720.189} C_VEL
LIN {X 0,Y 616.003,Z 1284.062,A -85,B 0,C 180,E1 28717.838,E2 28717.838} C_VEL
LIN {X 0,Y 615.937,Z 1288.645,A -85,B 0,C 180,E1 28715.965,E2 28715.965} C_VEL
LIN {X 0,Y 615.914,Z 1291.961,A -85,B 0,C 180,E1 28714.097,E2 28714.097} C_VEL
LIN {X 0,Y 615.904,Z 1294.042,A -85,B 0,C 180,E1 28712.234,E2 28712.234} C_VEL
LIN {X 0,Y 615.908,Z 1294.984,A -85,B 0,C 180,E1 28710.094,E2 28710.094} C_VEL
LIN {X 0,Y 615.907,Z 1294.13,A -85,B 0,C 180,E1 28707.861,E2 28707.861} C_VEL
LIN {X 0,Y 615.911,Z 1292.101,A -85,B 0,C 180,E1 28705.998,E2 28705.998} C_VEL
LIN {X 0,Y 615.927,Z 1289.028,A -85,B 0,C 180,E1 28704.225,E2 28704.225} C_VEL
LIN {X 0,Y 615.998,Z 1285.052,A -85,B 0,C 180,E1 28702.54,E2 28702.54} C_VEL
LIN {X 0,Y 616.088,Z 1280.012,A -85,B 0,C 180,E1 28700.85,E2 28700.85} C_VEL
LIN {X 0,Y 616.276,Z 1273.845,A -85,B 0,C 180,E1 28699.153,E2 28699.153} C_VEL
LIN {X 0,Y 616.565,Z 1266.044,A -85,B 0,C 180,E1 28697.355,E2 28697.355} C_VEL
LIN {X 0,Y 617.088,Z 1255.273,A -85,B 0,C 180,E1 28695.264,E2 28695.264} C_VEL
LIN {X 0,Y 617.752,Z 1243.426,A -85,B 0,C 180,E1 28693.354,E2 28693.354} C_VEL
LIN {X 0,Y 618.445,Z 1232.575,A -85,B 0,C 180,E1 28691.819,E2 28691.819} C_VEL
LIN {X 0,Y 619.256,Z 1221.083,A -85,B 0,C 180,E1 28690.377,E2 28690.377} C_VEL
LIN {X 0,Y 620.002,Z 1210.729,A -85,B 0,C 180,E1 28689.221,E2 28689.221} C_VEL
LIN {X 0,Y 620.966,Z 1196.837,A -85,B 0,C 180,E1 28687.867,E2 28687.867} C_VEL
LIN {X 0,Y 621.978,Z 1182.341,A -85,B 0,C 180,E1 28686.606,E2 28686.606} C_VEL
LIN {X 0,Y 623.303,Z 1164.491,A -85,B 0,C 180,E1 28685.226,E2 28685.226} C_VEL
LIN {X 0,Y 624.759,Z 1143.663,A -85,B 0,C 180,E1 28683.844,E2 28683.844} C_VEL
LIN {X 0,Y 626.277,Z 1122.288,A -85,B 0,C 180,E1 28682.627,E2 28682.627} C_VEL
LIN {X 0,Y 627.74,Z 1099.93,A -85,B 0,C 180,E1 28681.552,E2 28681.552} C_VEL
LIN {X 0,Y 629.221,Z 1076.705,A -85,B 0,C 180,E1 28680.62,E2 28680.62} C_VEL
LIN {X 0,Y 630.523,Z 1053.974,A -85,B 0,C 180,E1 28679.889,E2 28679.889} C_VEL
LIN {X 0,Y 631.71,Z 1031.06,A -85,B 0,C 180,E1 28679.301,E2 28679.301} C_VEL
LIN {X 0,Y 632.657,Z 1008.175,A -85,B 0,C 180,E1 28678.882,E2 28678.882} C_VEL
LIN {X 0,Y 633.721,Z 970.721,A -85,B 0,C 180,E1 28678.391,E2 28678.391} C_VEL
LIN {X 0,Y 634.364,Z 966.519,A -85,B 0,C 180,E1 28678.338,E2 28678.338} C_VEL
LIN {X 0,Y 639.803,Z 955.466,A -85,B 0,C 180,E1 28677.746,E2 28677.746} C_VEL
LIN {X 0,Y 650.38,Z 938.135,A -85,B 0,C 180,E1 28676.924,E2 28676.924} C_VEL
LIN {X 0,Y 659.072,Z 926.863,A -85,B 0,C 180,E1 28676.482,E2 28676.482} C_VEL
LIN {X 0,Y 671.213,Z 913.821,A -85,B 0,C 180,E1 28676.074,E2 28676.074} C_VEL
LIN {X 0,Y 686.691,Z 898.901,A -85,B 0,C 180,E1 28675.693,E2 28675.693} C_VEL
LIN {X 0,Y 674.505,Z 893.74,A -85,B 0,C 180,E1 28674.767,E2 28674.767} C_VEL
LIN {X 0,Y 663.455,Z 887.003,A -85,B 0,C 180,E1 28673.736,E2 28673.736} C_VEL
LIN {X 0,Y 654.668,Z 879.578,A -85,B 0,C 180,E1 28672.725,E2 28672.725} C_VEL
LIN {X 0,Y 646.748,Z 870.28,A -85,B 0,C 180,E1 28671.576,E2 28671.576} C_VEL
LIN {X 0,Y 640.366,Z 859.241,A -85,B 0,C 180,E1 28670.335,E2 28670.335} C_VEL
LIN {X 0,Y 635.841,Z 847.016,A -85,B 0,C 180,E1 28669.079,E2 28669.079} C_VEL
LIN {X 0,Y 633.162,Z 833.377,A -85,B 0,C 180,E1 28667.787,E2 28667.787} C_VEL
LIN {X 0,Y 632.234,Z 816.029,A -85,B 0,C 180,E1 28666.283,E2 28666.283} C_VEL
LIN {X 0,Y 634.926,Z 769.206,A -85,B 0,C 180,E1 28662.465,E2 28662.465} C_VEL
LIN {X 0,Y 637.266,Z 733.151,A -85,B 0,C 180,E1 28659.454,E2 28659.454} C_VEL
LIN {X 0,Y 639.483,Z 698.965,A -85,B 0,C 180,E1 28656.52,E2 28656.52} C_VEL
LIN {X 0,Y 641.501,Z 667.394,A -85,B 0,C 180,E1 28653.73,E2 28653.73} C_VEL
LIN {X 0,Y 632.589,Z 646.301,A -85,B 0,C 180,E1 28650.806,E2 28650.806} C_VEL
LIN {X 0,Y 624.245,Z 627.367,A -85,B 0,C 180,E1 28647.99,E2 28647.99} C_VEL
LIN {X 0,Y 618.385,Z 614.698,A -85,B 0,C 180,E1 28645.989,E2 28645.989} C_VEL
LIN {X 0,Y 617.01,Z 611.124,A -85,B 0,C 180,E1 28645.432,E2 28645.432} C_VEL
LIN {X 0,Y 617.007,Z 611.123,A -85,B 0,C 180,E1 28642.184,E2 28642.184} C_VEL
LIN {X 0,Y 617.003,Z 611.12,A -85,B 0,C 180,E1 28639.01,E2 28639.01} C_VEL
LIN {X 0,Y 616.999,Z 611.125,A -85,B 0,C 180,E1 28635.799,E2 28635.799} C_VEL
LIN {X 0,Y 616.998,Z 611.122,A -85,B 0,C 180,E1 28632.697,E2 28632.697} C_VEL
LIN {X 0,Y 616.998,Z 611.124,A -85,B 0,C 180,E1 28629.515,E2 28629.515} C_VEL
LIN {X 0,Y 616.998,Z 611.119,A -85,B 0,C 180,E1 28626.42,E2 28626.42} C_VEL
LIN {X 0,Y 616.998,Z 611.124,A -85,B 0,C 180,E1 28623.252,E2 28623.252} C_VEL
LIN {X 0,Y 617.002,Z 611.126,A -85,B 0,C 180,E1 28620.186,E2 28620.186} C_VEL
LIN {X 0,Y 616.998,Z 611.126,A -85,B 0,C 180,E1 28617.027,E2 28617.027} C_VEL
LIN {X 0,Y 617.008,Z 611.125,A -85,B 0,C 180,E1 28613.953,E2 28613.953} C_VEL
LIN {X 0,Y 616.999,Z 611.125,A -85,B 0,C 180,E1 28610.768,E2 28610.768} C_VEL
LIN {X 0,Y 617.011,Z 611.123,A -85,B 0,C 180,E1 28607.648,E2 28607.648} C_VEL
LIN {X 0,Y 617.005,Z 611.125,A -85,B 0,C 180,E1 28604.491,E2 28604.491} C_VEL
LIN {X 0,Y 617.014,Z 611.124,A -85,B 0,C 180,E1 28601.285,E2 28601.285} C_VEL
LIN {X 0,Y 617.001,Z 611.127,A -85,B 0,C 180,E1 28598.116,E2 28598.116} C_VEL
LIN {X 0,Y 617.017,Z 611.125,A -85,B 0,C 180,E1 28594.876,E2 28594.876} C_VEL
LIN {X 0,Y 617.008,Z 611.125,A -85,B 0,C 180,E1 28591.633,E2 28591.633} C_VEL
LIN {X 0,Y 617.02,Z 611.121,A -85,B 0,C 180,E1 28588.437,E2 28588.437} C_VEL
LIN {X 0,Y 617.011,Z 611.117,A -85,B 0,C 180,E1 28585.22,E2 28585.22} C_VEL
LIN {X 0,Y 617.013,Z 611.118,A -85,B 0,C 180,E1 28581.957,E2 28581.957} C_VEL
LIN {X 0,Y 617.007,Z 611.12,A -85,B 0,C 180,E1 28578.733,E2 28578.733} C_VEL
LIN {X 0,Y 617,Z 611.116,A -85,B 0,C 180,E1 28575.481,E2 28575.481} C_VEL
LIN {X 0,Y 616.999,Z 611.114,A -85,B 0,C 180,E1 28572.355,E2 28572.355} C_VEL
LIN {X 0,Y 616.998,Z 611.128,A -85,B 0,C 180,E1 28569.197,E2 28569.197} C_VEL
LIN {X 0,Y 617.002,Z 611.131,A -85,B 0,C 180,E1 28566.147,E2 28566.147} C_VEL
LIN {X 0,Y 617.012,Z 611.118,A -85,B 0,C 180,E1 28564.894,E2 28564.894} C_VEL
LIN {X 0,Y 615.998,Z 611.239,A -85,B 0,C 180,E1 28564.382,E2 28564.382} C_VEL
LIN {X 0,Y 612.54,Z 612.337,A -85,B 0,C 180,E1 28563.63,E2 28563.63} C_VEL
LIN {X 0,Y 610.827,Z 614.19,A -85,B 0,C 180,E1 28563.19,E2 28563.19} C_VEL
LIN {X 0,Y 610.577,Z 616.777,A -85,B 0,C 180,E1 28562.857,E2 28562.857} C_VEL
LIN {X 0,Y 610.713,Z 617.303,A -85,B 0,C 180,E1 28562.811,E2 28562.811} C_VEL
LIN {X 0,Y 618.298,Z 641.512,A -85,B 0,C 180,E1 28560.8,E2 28560.8} C_VEL
LIN {X 0,Y 617.482,Z 679.079,A -85,B 0,C 180,E1 28558.217,E2 28558.217} C_VEL
LIN {X 0,Y 616.276,Z 721.446,A -85,B 0,C 180,E1 28555.257,E2 28555.257} C_VEL
LIN {X 0,Y 614.81,Z 770.074,A -85,B 0,C 180,E1 28551.864,E2 28551.864} C_VEL
LIN {X 0,Y 613.638,Z 817.877,A -85,B 0,C 180,E1 28548.623,E2 28548.623} C_VEL
LIN {X 0,Y 613.37,Z 838.817,A -85,B 0,C 180,E1 28547.277,E2 28547.277} C_VEL
LIN {X 0,Y 614.166,Z 847.69,A -85,B 0,C 180,E1 28547.144,E2 28547.144} C_VEL
LIN {X 0,Y 612.945,Z 1008.2,A -85,B 0,C 180,E1 28545.22,E2 28545.22} C_VEL
LIN {X 0,Y 612.736,Z 1025.667,A -85,B 0,C 180,E1 28544.839,E2 28544.839} C_VEL
LIN {X 0,Y 612.383,Z 1041.643,A -85,B 0,C 180,E1 28544.32,E2 28544.32} C_VEL
LIN {X 0,Y 611.891,Z 1057.953,A -85,B 0,C 180,E1 28543.608,E2 28543.608} C_VEL
LIN {X 0,Y 611.333,Z 1073.182,A -85,B 0,C 180,E1 28542.755,E2 28542.755} C_VEL
LIN {X 0,Y 610.738,Z 1087.441,A -85,B 0,C 180,E1 28541.751,E2 28541.751} C_VEL
LIN {X 0,Y 610.174,Z 1099.888,A -85,B 0,C 180,E1 28540.67,E2 28540.67} C_VEL
LIN {X 0,Y 609.598,Z 1112.317,A -85,B 0,C 180,E1 28539.344,E2 28539.344} C_VEL
LIN {X 0,Y 609.153,Z 1122.368,A -85,B 0,C 180,E1 28538.019,E2 28538.019} C_VEL
LIN {X 0,Y 608.794,Z 1130.971,A -85,B 0,C 180,E1 28536.6,E2 28536.6} C_VEL
LIN {X 0,Y 608.539,Z 1138.146,A -85,B 0,C 180,E1 28535.089,E2 28535.089} C_VEL
LIN {X 0,Y 608.375,Z 1143.824,A -85,B 0,C 180,E1 28533.485,E2 28533.485} C_VEL
LIN {X 0,Y 608.278,Z 1147.696,A -85,B 0,C 180,E1 28531.883,E2 28531.883} C_VEL
LIN {X 0,Y 608.243,Z 1149.897,A -85,B 0,C 180,E1 28530.187,E2 28530.187} C_VEL
LIN {X 0,Y 608.226,Z 1150.31,A -85,B 0,C 180,E1 28528.492,E2 28528.492} C_VEL
LIN {X 0,Y 608.256,Z 1148.945,A -85,B 0,C 180,E1 28526.795,E2 28526.795} C_VEL
LIN {X 0,Y 608.323,Z 1145.901,A -85,B 0,C 180,E1 28525.19,E2 28525.19} C_VEL
LIN {X 0,Y 608.457,Z 1141.091,A -85,B 0,C 180,E1 28523.583,E2 28523.583} C_VEL
LIN {X 0,Y 608.673,Z 1134.388,A -85,B 0,C 180,E1 28521.972,E2 28521.972} C_VEL
LIN {X 0,Y 608.979,Z 1126.65,A -85,B 0,C 180,E1 28520.549,E2 28520.549} C_VEL
LIN {X 0,Y 609.398,Z 1116.822,A -85,B 0,C 180,E1 28519.123,E2 28519.123} C_VEL
LIN {X 0,Y 609.926,Z 1105.425,A -85,B 0,C 180,E1 28517.79,E2 28517.79} C_VEL
LIN {X 0,Y 610.496,Z 1093.194,A -85,B 0,C 180,E1 28516.625,E2 28516.625} C_VEL
LIN {X 0,Y 611.076,Z 1079.942,A -85,B 0,C 180,E1 28515.597,E2 28515.597} C_VEL
LIN {X 0,Y 611.636,Z 1065.509,A -85,B 0,C 180,E1 28514.693,E2 28514.693} C_VEL
LIN {X 0,Y 612.155,Z 1050.073,A -85,B 0,C 180,E1 28513.926,E2 28513.926} C_VEL
LIN {X 0,Y 612.59,Z 1033.711,A -85,B 0,C 180,E1 28513.304,E2 28513.304} C_VEL
LIN {X 0,Y 612.887,Z 1016.528,A -85,B 0,C 180,E1 28512.842,E2 28512.842} C_VEL
LIN {X 0,Y 613.028,Z 997.906,A -85,B 0,C 180,E1 28512.536,E2 28512.536} C_VEL
LIN {X 0,Y 614.008,Z 843.39,A -85,B 0,C 180,E1 28510.697,E2 28510.697} C_VEL
LIN {X 0,Y 613.335,Z 838.121,A -85,B 0,C 180,E1 28510.602,E2 28510.602} C_VEL
LIN {X 0,Y 614.331,Z 790.275,A -85,B 0,C 180,E1 28507.41,E2 28507.41} C_VEL
LIN {X 0,Y 615.679,Z 744.029,A -85,B 0,C 180,E1 28504.198,E2 28504.198} C_VEL
LIN {X 0,Y 617.049,Z 701.08,A -85,B 0,C 180,E1 28501.178,E2 28501.178} C_VEL
LIN {X 0,Y 618.18,Z 659.786,A -85,B 0,C 180,E1 28498.298,E2 28498.298} C_VEL
LIN {X 0,Y 618.468,Z 641.541,A -85,B 0,C 180,E1 28497.043,E2 28497.043} C_VEL
LIN {X 0,Y 610.959,Z 617.874,A -85,B 0,C 180,E1 28495.053,E2 28495.053} C_VEL
LIN {X 0,Y 609.074,Z 612.11,A -85,B 0,C 180,E1 28494.555,E2 28494.555} C_VEL
LIN {X 0,Y 609.076,Z 612.11,A -85,B 0,C 180,E1 28491.392,E2 28491.392} C_VEL
LIN {X 0,Y 609.068,Z 612.11,A -85,B 0,C 180,E1 28488.187,E2 28488.187} C_VEL
LIN {X 0,Y 609.063,Z 612.111,A -85,B 0,C 180,E1 28484.962,E2 28484.962} C_VEL
LIN {X 0,Y 609.07,Z 612.112,A -85,B 0,C 180,E1 28481.799,E2 28481.799} C_VEL
LIN {X 0,Y 609.058,Z 612.111,A -85,B 0,C 180,E1 28478.606,E2 28478.606} C_VEL
LIN {X 0,Y 609.074,Z 612.11,A -85,B 0,C 180,E1 28475.416,E2 28475.416} C_VEL
LIN {X 0,Y 609.086,Z 612.217,A -85,B 0,C 180,E1 28474.892,E2 28474.892} C_VEL
LIN {X 0,Y 610.524,Z 615.827,A -85,B 0,C 180,E1 28474.404,E2 28474.404} C_VEL
LIN {X 0,Y 612.054,Z 619.387,A -85,B 0,C 180,E1 28473.952,E2 28473.952} C_VEL
LIN {X 0,Y 627.175,Z 642.227,A -85,B 0,C 180,E1 28472.522,E2 28472.522} C_VEL
LIN {X 0,Y 630.898,Z 649.01,A -85,B 0,C 180,E1 28472.167,E2 28472.167} C_VEL
LIN {X 0,Y 626.078,Z 872.622,A -85,B 0,C 180,E1 28469.162,E2 28469.162} C_VEL
LIN {X 0,Y 624.608,Z 955.233,A -85,B 0,C 180,E1 28468.063,E2 28468.063} C_VEL
LIN {X 0,Y 623.815,Z 978.136,A -85,B 0,C 180,E1 28467.589,E2 28467.589} C_VEL
LIN {X 0,Y 622.811,Z 1001.123,A -85,B 0,C 180,E1 28466.948,E2 28466.948} C_VEL
LIN {X 0,Y 621.673,Z 1022.16,A -85,B 0,C 180,E1 28466.195,E2 28466.195} C_VEL
LIN {X 0,Y 620.239,Z 1043.821,A -85,B 0,C 180,E1 28465.245,E2 28465.245} C_VEL
LIN {X 0,Y 618.823,Z 1063.839,A -85,B 0,C 180,E1 28464.194,E2 28464.194} C_VEL
LIN {X 0,Y 617.279,Z 1083.387,A -85,B 0,C 180,E1 28462.978,E2 28462.978} C_VEL
LIN {X 0,Y 615.566,Z 1103.803,A -85,B 0,C 180,E1 28461.487,E2 28461.487} C_VEL
LIN {X 0,Y 614.177,Z 1120.231,A -85,B 0,C 180,E1 28460.091,E2 28460.091} C_VEL
LIN {X 0,Y 612.818,Z 1136.031,A -85,B 0,C 180,E1 28458.552,E2 28458.552} C_VEL
LIN {X 0,Y 611.505,Z 1152.311,A -85,B 0,C 180,E1 28456.725,E2 28456.725} C_VEL
LIN {X 0,Y 610.411,Z 1166.232,A -85,B 0,C 180,E1 28454.881,E2 28454.881} C_VEL
LIN {X 0,Y 609.636,Z 1177.514,A -85,B 0,C 180,E1 28453.178,E2 28453.178} C_VEL
LIN {X 0,Y 609.113,Z 1186.467,A -85,B 0,C 180,E1 28451.649,E2 28451.649} C_VEL
LIN {X 0,Y 608.673,Z 1194.783,A -85,B 0,C 180,E1 28450.028,E2 28450.028} C_VEL
LIN {X 0,Y 608.366,Z 1202.27,A -85,B 0,C 180,E1 28448.336,E2 28448.336} C_VEL
LIN {X 0,Y 608.153,Z 1208.731,A -85,B 0,C 180,E1 28446.609,E2 28446.609} C_VEL
LIN {X 0,Y 608.028,Z 1213.989,A -85,B 0,C 180,E1 28444.906,E2 28444.906} C_VEL
LIN {X 0,Y 607.955,Z 1218.176,A -85,B 0,C 180,E1 28443.206,E2 28443.206} C_VEL
LIN {X 0,Y 607.916,Z 1221.345,A -85,B 0,C 180,E1 28441.508,E2 28441.508} C_VEL
LIN {X 0,Y 607.907,Z 1223.504,A -85,B 0,C 180,E1 28439.812,E2 28439.812} C_VEL
LIN {X 0,Y 607.911,Z 1224.7,A -85,B 0,C 180,E1 28438.021,E2 28438.021} C_VEL
LIN {X 0,Y 607.913,Z 1224.821,A -85,B 0,C 180,E1 28436.322,E2 28436.322} C_VEL
LIN {X 0,Y 607.911,Z 1223.968,A -85,B 0,C 180,E1 28434.62,E2 28434.62} C_VEL
LIN {X 0,Y 607.923,Z 1221.971,A -85,B 0,C 180,E1 28432.819,E2 28432.819} C_VEL
LIN {X 0,Y 607.943,Z 1219.025,A -85,B 0,C 180,E1 28431.106,E2 28431.106} C_VEL
LIN {X 0,Y 607.996,Z 1215.018,A -85,B 0,C 180,E1 28429.386,E2 28429.386} C_VEL
LIN {X 0,Y 608.123,Z 1209.922,A -85,B 0,C 180,E1 28427.658,E2 28427.658} C_VEL
LIN {X 0,Y 608.307,Z 1203.66,A -85,B 0,C 180,E1 28425.92,E2 28425.92} C_VEL
LIN {X 0,Y 608.595,Z 1196.609,A -85,B 0,C 180,E1 28424.271,E2 28424.271} C_VEL
LIN {X 0,Y 608.976,Z 1188.891,A -85,B 0,C 180,E1 28422.711,E2 28422.711} C_VEL
LIN {X 0,Y 609.486,Z 1180.037,A -85,B 0,C 180,E1 28421.144,E2 28421.144} C_VEL
LIN {X 0,Y 610.102,Z 1170.33,A -85,B 0,C 180,E1 28419.628,E2 28419.628} C_VEL
LIN {X 0,Y 610.906,Z 1159.624,A -85,B 0,C 180,E1 28418.131,E2 28418.131} C_VEL
LIN {X 0,Y 611.801,Z 1148.07,A -85,B 0,C 180,E1 28416.702,E2 28416.702} C_VEL
LIN {X 0,Y 612.953,Z 1133.95,A -85,B 0,C 180,E1 28415.162,E2 28415.162} C_VEL
LIN {X 0,Y 614.372,Z 1116.49,A -85,B 0,C 180,E1 28413.526,E2 28413.526} C_VEL
LIN {X 0,Y 615.734,Z 1098.86,A -85,B 0,C 180,E1 28412.116,E2 28412.116} C_VEL
LIN {X 0,Y 617.032,Z 1081.447,A -85,B 0,C 180,E1 28410.912,E2 28410.912} C_VEL
LIN {X 0,Y 618.279,Z 1062.589,A -85,B 0,C 180,E1 28409.804,E2 28409.804} C_VEL
LIN {X 0,Y 619.441,Z 1042.81,A -85,B 0,C 180,E1 28408.818,E2 28408.818} C_VEL
LIN {X 0,Y 620.443,Z 1022.172,A -85,B 0,C 180,E1 28407.98,E2 28407.98} C_VEL
LIN {X 0,Y 621.274,Z 1000.596,A -85,B 0,C 180,E1 28407.269,E2 28407.269} C_VEL
LIN {X 0,Y 621.835,Z 979.067,A -85,B 0,C 180,E1 28406.733,E2 28406.733} C_VEL
LIN {X 0,Y 622.25,Z 955.048,A -85,B 0,C 180,E1 28406.315,E2 28406.315} C_VEL
LIN {X 0,Y 623.674,Z 749.836,A -85,B 0,C 180,E1 28403.963,E2 28403.963} C_VEL
LIN {X 0,Y 624.865,Z 650.586,A -85,B 0,C 180,E1 28402.709,E2 28402.709} C_VEL
LIN {X 0,Y 625.4,Z 651.836,A -85,B 0,C 180,E1 28401.659,E2 28401.659} C_VEL
LIN {X 0,Y 626.153,Z 654.232,A -85,B 0,C 180,E1 28400.723,E2 28400.723} C_VEL
LIN {X 0,Y 621.031,Z 664.486,A -85,B 0,C 180,E1 28399.46,E2 28399.46} C_VEL
LIN {X 0,Y 617.054,Z 676.596,A -85,B 0,C 180,E1 28398.194,E2 28398.194} C_VEL
LIN {X 0,Y 614.075,Z 690.93,A -85,B 0,C 180,E1 28396.911,E2 28396.911} C_VEL
LIN {X 0,Y 611.794,Z 709.486,A -85,B 0,C 180,E1 28395.481,E2 28395.481} C_VEL
LIN {X 0,Y 610.106,Z 735.073,A -85,B 0,C 180,E1 28393.758,E2 28393.758} C_VEL
LIN {X 0,Y 609.308,Z 771.549,A -85,B 0,C 180,E1 28391.528,E2 28391.528} C_VEL
LIN {X 0,Y 610.705,Z 793.877,A -85,B 0,C 180,E1 28390.193,E2 28390.193} C_VEL
LIN {X 0,Y 613.794,Z 812.363,A -85,B 0,C 180,E1 28389.083,E2 28389.083} C_VEL
LIN {X 0,Y 618.344,Z 828.118,A -85,B 0,C 180,E1 28388.13,E2 28388.13} C_VEL
LIN {X 0,Y 625.01,Z 843.771,A -85,B 0,C 180,E1 28387.183,E2 28387.183} C_VEL
LIN {X 0,Y 633.115,Z 857.757,A -85,B 0,C 180,E1 28386.346,E2 28386.346} C_VEL
LIN {X 0,Y 642.981,Z 870.783,A -85,B 0,C 180,E1 28385.579,E2 28385.579} C_VEL
LIN {X 0,Y 654.602,Z 882.822,A -85,B 0,C 180,E1 28384.889,E2 28384.889} C_VEL
LIN {X 0,Y 667.065,Z 893.155,A -85,B 0,C 180,E1 28384.318,E2 28384.318} C_VEL
LIN {X 0,Y 673.275,Z 897.653,A -85,B 0,C 180,E1 28384.073,E2 28384.073} C_VEL
LIN {X 0,Y 657.489,Z 910.465,A -85,B 0,C 180,E1 28383.403,E2 28383.403} C_VEL
LIN {X 0,Y 646.217,Z 921.804,A -85,B 0,C 180,E1 28382.79,E2 28382.79} C_VEL
LIN {X 0,Y 638.003,Z 932.51,A -85,B 0,C 180,E1 28382.199,E2 28382.199} C_VEL
LIN {X 0,Y 627.38,Z 950.24,A -85,B 0,C 180,E1 28381.201,E2 28381.201} C_VEL
LIN {X 0,Y 622.979,Z 966.678,A -85,B 0,C 180,E1 28381.143,E2 28381.143} C_VEL
LIN {X 0,Y 622.031,Z 976.885,A -85,B 0,C 180,E1 28381.053,E2 28381.053} C_VEL
LIN {X 0,Y 621.539,Z 1006.485,A -85,B 0,C 180,E1 28380.638,E2 28380.638} C_VEL
LIN {X 0,Y 620.633,Z 1034.543,A -85,B 0,C 180,E1 28380.073,E2 28380.073} C_VEL
LIN {X 0,Y 619.696,Z 1060.839,A -85,B 0,C 180,E1 28379.375,E2 28379.375} C_VEL
LIN {X 0,Y 618.684,Z 1087.014,A -85,B 0,C 180,E1 28378.502,E2 28378.502} C_VEL
LIN {X 0,Y 617.62,Z 1110.871,A -85,B 0,C 180,E1 28377.531,E2 28377.531} C_VEL
LIN {X 0,Y 616.551,Z 1133.15,A -85,B 0,C 180,E1 28376.447,E2 28376.447} C_VEL
LIN {X 0,Y 615.545,Z 1152.301,A -85,B 0,C 180,E1 28375.364,E2 28375.364} C_VEL
LIN {X 0,Y 614.429,Z 1171.959,A -85,B 0,C 180,E1 28374.084,E2 28374.084} C_VEL
LIN {X 0,Y 613.236,Z 1191.4,A -85,B 0,C 180,E1 28372.585,E2 28372.585} C_VEL
LIN {X 0,Y 612.334,Z 1205.814,A -85,B 0,C 180,E1 28371.305,E2 28371.305} C_VEL
LIN {X 0,Y 611.549,Z 1218.038,A -85,B 0,C 180,E1 28370.082,E2 28370.082} C_VEL
LIN {X 0,Y 610.841,Z 1229.282,A -85,B 0,C 180,E1 28368.813,E2 28368.813} C_VEL
LIN {X 0,Y 610.173,Z 1239.525,A -85,B 0,C 180,E1 28367.452,E2 28367.452} C_VEL
LIN {X 0,Y 609.447,Z 1250.669,A -85,B 0,C 180,E1 28365.707,E2 28365.707} C_VEL
LIN {X 0,Y 608.927,Z 1259.832,A -85,B 0,C 180,E1 28364.066,E2 28364.066} C_VEL
LIN {X 0,Y 608.55,Z 1267.769,A -85,B 0,C 180,E1 28362.431,E2 28362.431} C_VEL
LIN {X 0,Y 608.273,Z 1274.938,A -85,B 0,C 180,E1 28360.706,E2 28360.706} C_VEL
LIN {X 0,Y 608.08,Z 1280.921,A -85,B 0,C 180,E1 28358.988,E2 28358.988} C_VEL
LIN {X 0,Y 607.983,Z 1286.037,A -85,B 0,C 180,E1 28357.181,E2 28357.181} C_VEL
LIN {X 0,Y 607.915,Z 1290.863,A -85,B 0,C 180,E1 28354.908,E2 28354.908} C_VEL
LIN {X 0,Y 607.899,Z 1293.636,A -85,B 0,C 180,E1 28352.735,E2 28352.735} C_VEL
LIN {X 0,Y 607.904,Z 1294.777,A -85,B 0,C 180,E1 28350.849,E2 28350.849} C_VEL
LIN {X 0,Y 607.904,Z 1294.773,A -85,B 0,C 180,E1 28349.153,E2 28349.153} C_VEL
LIN {X 0,Y 607.897,Z 1293.713,A -85,B 0,C 180,E1 28347.362,E2 28347.362} C_VEL
LIN {X 0,Y 607.908,Z 1291.406,A -85,B 0,C 180,E1 28345.473,E2 28345.473} C_VEL
LIN {X 0,Y 607.953,Z 1287.467,A -85,B 0,C 180,E1 28343.39,E2 28343.39} C_VEL
LIN {X 0,Y 608.074,Z 1281.253,A -85,B 0,C 180,E1 28341.11,E2 28341.11} C_VEL
LIN {X 0,Y 608.273,Z 1274.957,A -85,B 0,C 180,E1 28339.297,E2 28339.297} C_VEL
LIN {X 0,Y 608.55,Z 1267.783,A -85,B 0,C 180,E1 28337.572,E2 28337.572} C_VEL
LIN {X 0,Y 608.926,Z 1259.844,A -85,B 0,C 180,E1 28335.936,E2 28335.936} C_VEL
LIN {X 0,Y 609.444,Z 1250.679,A -85,B 0,C 180,E1 28334.295,E2 28334.295} C_VEL
LIN {X 0,Y 610.075,Z 1240.824,A -85,B 0,C 180,E1 28332.745,E2 28332.745} C_VEL
LIN {X 0,Y 610.639,Z 1232.4,A -85,B 0,C 180,E1 28331.579,E2 28331.579} C_VEL
LIN {X 0,Y 611.458,Z 1220.393,A -85,B 0,C 180,E1 28330.117,E2 28330.117} C_VEL
LIN {X 0,Y 612.392,Z 1207.304,A -85,B 0,C 180,E1 28328.699,E2 28328.699} C_VEL
LIN {X 0,Y 613.488,Z 1192.547,A -85,B 0,C 180,E1 28327.279,E2 28327.279} C_VEL
LIN {X 0,Y 614.944,Z 1173.542,A -85,B 0,C 180,E1 28325.672,E2 28325.672} C_VEL
LIN {X 0,Y 616.521,Z 1152.781,A -85,B 0,C 180,E1 28324.174,E2 28324.174} C_VEL
LIN {X 0,Y 618.152,Z 1131.102,A -85,B 0,C 180,E1 28322.83,E2 28322.83} C_VEL
LIN {X 0,Y 619.797,Z 1108.699,A -85,B 0,C 180,E1 28321.652,E2 28321.652} C_VEL
LIN {X 0,Y 621.513,Z 1083.753,A -85,B 0,C 180,E1 28320.563,E2 28320.563} C_VEL
LIN {X 0,Y 623.046,Z 1060.609,A -85,B 0,C 180,E1 28319.742,E2 28319.742} C_VEL
LIN {X 0,Y 624.425,Z 1036.695,A -85,B 0,C 180,E1 28319.078,E2 28319.078} C_VEL
LIN {X 0,Y 625.679,Z 1011.752,A -85,B 0,C 180,E1 28318.559,E2 28318.559} C_VEL
LIN {X 0,Y 626.347,Z 985.235,A -85,B 0,C 180,E1 28318.187,E2 28318.187} C_VEL
LIN {X 0,Y 627.136,Z 969.104,A -85,B 0,C 180,E1 28317.986,E2 28317.986} C_VEL
LIN {X 0,Y 627.759,Z 965.095,A -85,B 0,C 180,E1 28317.943,E2 28317.943} C_VEL
LIN {X 0,Y 633.494,Z 953.675,A -85,B 0,C 180,E1 28317.332,E2 28317.332} C_VEL
LIN {X 0,Y 644.149,Z 936.345,A -85,B 0,C 180,E1 28316.509,E2 28316.509} C_VEL
LIN {X 0,Y 653.391,Z 924.374,A -85,B 0,C 180,E1 28316.04,E2 28316.04} C_VEL
LIN {X 0,Y 665.836,Z 910.992,A -85,B 0,C 180,E1 28315.625,E2 28315.625} C_VEL
LIN {X 0,Y 674.876,Z 902.076,A -85,B 0,C 180,E1 28315.389,E2 28315.389} C_VEL
LIN {X 0,Y 663.69,Z 896.342,A -85,B 0,C 180,E1 28314.444,E2 28314.444} C_VEL
LIN {X 0,Y 652.895,Z 888.653,A -85,B 0,C 180,E1 28313.327,E2 28313.327} C_VEL
LIN {X 0,Y 644.082,Z 879.865,A -85,B 0,C 180,E1 28312.18,E2 28312.18} C_VEL
LIN {X 0,Y 636.977,Z 869.872,A -85,B 0,C 180,E1 28310.989,E2 28310.989} C_VEL
LIN {X 0,Y 631.285,Z 858,A -85,B 0,C 180,E1 28309.698,E2 28309.698} C_VEL
LIN {X 0,Y 627.438,Z 844.734,A -85,B 0,C 180,E1 28308.366,E2 28308.366} C_VEL
LIN {X 0,Y 625.476,Z 829.779,A -85,B 0,C 180,E1 28306.994,E2 28306.994} C_VEL
LIN {X 0,Y 625.426,Z 811.37,A -85,B 0,C 180,E1 28305.427,E2 28305.427} C_VEL
LIN {X 0,Y 628.008,Z 772.182,A -85,B 0,C 180,E1 28302.214,E2 28302.214} C_VEL
LIN {X 0,Y 630.406,Z 737.07,A -85,B 0,C 180,E1 28299.261,E2 28299.261} C_VEL
LIN {X 0,Y 632.761,Z 702.88,A -85,B 0,C 180,E1 28296.306,E2 28296.306} C_VEL
LIN {X 0,Y 634.927,Z 671.401,A -85,B 0,C 180,E1 28293.503,E2 28293.503} C_VEL
LIN {X 0,Y 626.2,Z 650.755,A -85,B 0,C 180,E1 28290.614,E2 28290.614} C_VEL
LIN {X 0,Y 618.156,Z 632.413,A -85,B 0,C 180,E1 28287.87,E2 28287.87} C_VEL
LIN {X 0,Y 612.03,Z 619.26,A -85,B 0,C 180,E1 28285.758,E2 28285.758} C_VEL
LIN {X 0,Y 610.505,Z 615.794,A -85,B 0,C 180,E1 28285.203,E2 28285.203} C_VEL
LIN {X 0,Y 609.089,Z 612.268,A -85,B 0,C 180,E1 28284.644,E2 28284.644} C_VEL
LIN {X 0,Y 609.076,Z 612.113,A -85,B 0,C 180,E1 28281.374,E2 28281.374} C_VEL
LIN {X 0,Y 609.078,Z 612.114,A -85,B 0,C 180,E1 28278.107,E2 28278.107} C_VEL
LIN {X 0,Y 609.081,Z 612.109,A -85,B 0,C 180,E1 28274.839,E2 28274.839} C_VEL
LIN {X 0,Y 609.073,Z 612.114,A -85,B 0,C 180,E1 28271.65,E2 28271.65} C_VEL
LIN {X 0,Y 609.077,Z 612.109,A -85,B 0,C 180,E1 28268.401,E2 28268.401} C_VEL
LIN {X 0,Y 609.07,Z 612.114,A -85,B 0,C 180,E1 28265.18,E2 28265.18} C_VEL
LIN {X 0,Y 609.077,Z 612.11,A -85,B 0,C 180,E1 28261.882,E2 28261.882} C_VEL
LIN {X 0,Y 609.07,Z 612.108,A -85,B 0,C 180,E1 28258.589,E2 28258.589} C_VEL
LIN {X 0,Y 609.073,Z 612.11,A -85,B 0,C 180,E1 28255.292,E2 28255.292} C_VEL
LIN {X 0,Y 609.072,Z 612.111,A -85,B 0,C 180,E1 28252.074,E2 28252.074} C_VEL
LIN {X 0,Y 609.064,Z 612.112,A -85,B 0,C 180,E1 28248.83,E2 28248.83} C_VEL
LIN {X 0,Y 609.062,Z 612.112,A -85,B 0,C 180,E1 28245.647,E2 28245.647} C_VEL
LIN {X 0,Y 609.062,Z 612.113,A -85,B 0,C 180,E1 28242.513,E2 28242.513} C_VEL
LIN {X 0,Y 609.06,Z 612.112,A -85,B 0,C 180,E1 28239.346,E2 28239.346} C_VEL
LIN {X 0,Y 609.061,Z 612.11,A -85,B 0,C 180,E1 28236.283,E2 28236.283} C_VEL
LIN {X 0,Y 609.062,Z 612.107,A -85,B 0,C 180,E1 28233.162,E2 28233.162} C_VEL
LIN {X 0,Y 609.063,Z 612.111,A -85,B 0,C 180,E1 28230.061,E2 28230.061} C_VEL
LIN {X 0,Y 609.071,Z 612.114,A -85,B 0,C 180,E1 28226.973,E2 28226.973} C_VEL
LIN {X 0,Y 609.063,Z 612.116,A -85,B 0,C 180,E1 28223.771,E2 28223.771} C_VEL
LIN {X 0,Y 609.075,Z 612.111,A -85,B 0,C 180,E1 28220.641,E2 28220.641} C_VEL
LIN {X 0,Y 609.063,Z 612.096,A -85,B 0,C 180,E1 28217.484,E2 28217.484} C_VEL
LIN {X 0,Y 609.076,Z 612.114,A -85,B 0,C 180,E1 28214.294,E2 28214.294} C_VEL
LIN {X 0,Y 609.059,Z 612.102,A -85,B 0,C 180,E1 28211.045,E2 28211.045} C_VEL
LIN {X 0,Y 609.077,Z 612.102,A -85,B 0,C 180,E1 28207.848,E2 28207.848} C_VEL
LIN {X 0,Y 609.065,Z 612.104,A -85,B 0,C 180,E1 28204.61,E2 28204.61} C_VEL
LIN {X 0,Y 609.079,Z 612.173,A -85,B 0,C 180,E1 28203.235,E2 28203.235} C_VEL
LIN {X 0,Y 610.713,Z 617.303,A -85,B 0,C 180,E1 28202.811,E2 28202.811} C_VEL
LIN {X 0,Y 611.911,Z 624.147,A -85,B 0,C 180,E1 28202.293,E2 28202.293} C_VEL
LIN {X 0,Y 611.635,Z 635.097,A -85,B 0,C 180,E1 28201.566,E2 28201.566} C_VEL
LIN {X 0,Y 610.881,Z 646.149,A -85,B 0,C 180,E1 28200.844,E2 28200.844} C_VEL
LIN {X 0,Y 609.829,Z 690.024,A -85,B 0,C 180,E1 28197.804,E2 28197.804} C_VEL
LIN {X 0,Y 608.354,Z 736.607,A -85,B 0,C 180,E1 28194.518,E2 28194.518} C_VEL
LIN {X 0,Y 606.909,Z 783.486,A -85,B 0,C 180,E1 28191.249,E2 28191.249} C_VEL
LIN {X 0,Y 605.883,Z 828.405,A -85,B 0,C 180,E1 28188.222,E2 28188.222} C_VEL
LIN {X 0,Y 605.791,Z 839.696,A -85,B 0,C 180,E1 28187.51,E2 28187.51} C_VEL
LIN {X 0,Y 606.581,Z 848.439,A -85,B 0,C 180,E1 28187.377,E2 28187.377} C_VEL
LIN {X 0,Y 605.289,Z 1009.249,A -85,B 0,C 180,E1 28185.425,E2 28185.425} C_VEL
LIN {X 0,Y 605.073,Z 1026.695,A -85,B 0,C 180,E1 28185.039,E2 28185.039} C_VEL
LIN {X 0,Y 604.686,Z 1043.324,A -85,B 0,C 180,E1 28184.487,E2 28184.487} C_VEL
LIN {X 0,Y 604.154,Z 1060.149,A -85,B 0,C 180,E1 28183.732,E2 28183.732} C_VEL
LIN {X 0,Y 603.587,Z 1074.823,A -85,B 0,C 180,E1 28182.888,E2 28182.888} C_VEL
LIN {X 0,Y 602.953,Z 1088.994,A -85,B 0,C 180,E1 28181.865,E2 28181.865} C_VEL
LIN {X 0,Y 602.334,Z 1101.918,A -85,B 0,C 180,E1 28180.713,E2 28180.713} C_VEL
LIN {X 0,Y 601.772,Z 1113.36,A -85,B 0,C 180,E1 28179.467,E2 28179.467} C_VEL
LIN {X 0,Y 601.296,Z 1123.396,A -85,B 0,C 180,E1 28178.124,E2 28178.124} C_VEL
LIN {X 0,Y 600.909,Z 1131.983,A -85,B 0,C 180,E1 28176.687,E2 28176.687} C_VEL
LIN {X 0,Y 600.631,Z 1139.146,A -85,B 0,C 180,E1 28175.156,E2 28175.156} C_VEL
LIN {X 0,Y 600.45,Z 1144.814,A -85,B 0,C 180,E1 28173.531,E2 28173.531} C_VEL
LIN {X 0,Y 600.342,Z 1148.671,A -85,B 0,C 180,E1 28171.908,E2 28171.908} C_VEL
LIN {X 0,Y 600.301,Z 1150.859,A -85,B 0,C 180,E1 28170.19,E2 28170.19} C_VEL
LIN {X 0,Y 600.283,Z 1151.26,A -85,B 0,C 180,E1 28168.472,E2 28168.472} C_VEL
LIN {X 0,Y 600.318,Z 1149.882,A -85,B 0,C 180,E1 28166.752,E2 28166.752} C_VEL
LIN {X 0,Y 600.394,Z 1146.822,A -85,B 0,C 180,E1 28165.126,E2 28165.126} C_VEL
LIN {X 0,Y 600.545,Z 1142,A -85,B 0,C 180,E1 28163.498,E2 28163.498} C_VEL
LIN {X 0,Y 600.786,Z 1135.284,A -85,B 0,C 180,E1 28161.866,E2 28161.866} C_VEL
LIN {X 0,Y 601.119,Z 1127.529,A -85,B 0,C 180,E1 28160.424,E2 28160.424} C_VEL
LIN {X 0,Y 601.573,Z 1117.681,A -85,B 0,C 180,E1 28158.979,E2 28158.979} C_VEL
LIN {X 0,Y 602.141,Z 1106.267,A -85,B 0,C 180,E1 28157.63,E2 28157.63} C_VEL
LIN {X 0,Y 602.759,Z 1093.819,A -85,B 0,C 180,E1 28156.433,E2 28156.433} C_VEL
LIN {X 0,Y 603.391,Z 1080.012,A -85,B 0,C 180,E1 28155.361,E2 28155.361} C_VEL
LIN {X 0,Y 604.027,Z 1064.469,A -85,B 0,C 180,E1 28154.394,E2 28154.394} C_VEL
LIN {X 0,Y 604.582,Z 1048.481,A -85,B 0,C 180,E1 28153.615,E2 28153.615} C_VEL
LIN {X 0,Y 605.008,Z 1031.645,A -85,B 0,C 180,E1 28153.005,E2 28153.005} C_VEL
LIN {X 0,Y 605.288,Z 1013.689,A -85,B 0,C 180,E1 28152.553,E2 28152.553} C_VEL
LIN {X 0,Y 605.422,Z 993.603,A -85,B 0,C 180,E1 28152.258,E2 28152.258} C_VEL
LIN {X 0,Y 606.444,Z 844.123,A -85,B 0,C 180,E1 28150.456,E2 28150.456} C_VEL
LIN {X 0,Y 605.78,Z 838.975,A -85,B 0,C 180,E1 28150.36,E2 28150.36} C_VEL
LIN {X 0,Y 606.83,Z 790.519,A -85,B 0,C 180,E1 28147.115,E2 28147.115} C_VEL
LIN {X 0,Y 608.271,Z 743.584,A -85,B 0,C 180,E1 28143.836,E2 28143.836} C_VEL
LIN {X 0,Y 609.707,Z 699.866,A -85,B 0,C 180,E1 28140.743,E2 28140.743} C_VEL
LIN {X 0,Y 610.848,Z 660.279,A -85,B 0,C 180,E1 28137.97,E2 28137.97} C_VEL
LIN {X 0,Y 611.048,Z 643.915,A -85,B 0,C 180,E1 28136.833,E2 28136.833} C_VEL
LIN {X 0,Y 603.807,Z 621.115,A -85,B 0,C 180,E1 28134.891,E2 28134.891} C_VEL
LIN {X 0,Y 601.121,Z 613.092,A -85,B 0,C 180,E1 28134.192,E2 28134.192} C_VEL
LIN {X 0,Y 601.137,Z 613.089,A -85,B 0,C 180,E1 28130.967,E2 28130.967} C_VEL
LIN {X 0,Y 601.12,Z 613.102,A -85,B 0,C 180,E1 28127.777,E2 28127.777} C_VEL
LIN {X 0,Y 601.124,Z 613.098,A -85,B 0,C 180,E1 28124.583,E2 28124.583} C_VEL
LIN {X 0,Y 601.141,Z 613.103,A -85,B 0,C 180,E1 28121.326,E2 28121.326} C_VEL
LIN {X 0,Y 601.133,Z 613.101,A -85,B 0,C 180,E1 28118.105,E2 28118.105} C_VEL
LIN {X 0,Y 601.167,Z 613.306,A -85,B 0,C 180,E1 28115.543,E2 28115.543} C_VEL
LIN {X 0,Y 602.452,Z 616.607,A -85,B 0,C 180,E1 28115.091,E2 28115.091} C_VEL
LIN {X 0,Y 604.539,Z 621.246,A -85,B 0,C 180,E1 28114.482,E2 28114.482} C_VEL
LIN {X 0,Y 620.875,Z 645.821,A -85,B 0,C 180,E1 28112.896,E2 28112.896} C_VEL
LIN {X 0,Y 624.355,Z 652.003,A -85,B 0,C 180,E1 28112.559,E2 28112.559} C_VEL
LIN {X 0,Y 619.066,Z 879.41,A -85,B 0,C 180,E1 28109.45,E2 28109.45} C_VEL
LIN {X 0,Y 617.567,Z 956.433,A -85,B 0,C 180,E1 28108.402,E2 28108.402} C_VEL
LIN {X 0,Y 616.725,Z 979.685,A -85,B 0,C 180,E1 28107.911,E2 28107.911} C_VEL
LIN {X 0,Y 615.627,Z 1003.271,A -85,B 0,C 180,E1 28107.233,E2 28107.233} C_VEL
LIN {X 0,Y 614.452,Z 1023.916,A -85,B 0,C 180,E1 28106.48,E2 28106.48} C_VEL
LIN {X 0,Y 612.933,Z 1045.511,A -85,B 0,C 180,E1 28105.51,E2 28105.51} C_VEL
LIN {X 0,Y 611.381,Z 1066.362,A -85,B 0,C 180,E1 28104.391,E2 28104.391} C_VEL
LIN {X 0,Y 609.713,Z 1086.119,A -85,B 0,C 180,E1 28103.127,E2 28103.127} C_VEL
LIN {X 0,Y 608.017,Z 1105.222,A -85,B 0,C 180,E1 28101.696,E2 28101.696} C_VEL
LIN {X 0,Y 606.565,Z 1121.552,A -85,B 0,C 180,E1 28100.286,E2 28100.286} C_VEL
LIN {X 0,Y 605.033,Z 1138.456,A -85,B 0,C 180,E1 28098.6,E2 28098.6} C_VEL
LIN {X 0,Y 603.58,Z 1155.128,A -85,B 0,C 180,E1 28096.654,E2 28096.654} C_VEL
LIN {X 0,Y 602.589,Z 1167.324,A -85,B 0,C 180,E1 28095.002,E2 28095.002} C_VEL
LIN {X 0,Y 601.786,Z 1177.972,A -85,B 0,C 180,E1 28093.353,E2 28093.353} C_VEL
LIN {X 0,Y 601.209,Z 1186.746,A -85,B 0,C 180,E1 28091.804,E2 28091.804} C_VEL
LIN {X 0,Y 600.709,Z 1195.424,A -85,B 0,C 180,E1 28090.066,E2 28090.066} C_VEL
LIN {X 0,Y 600.395,Z 1202.582,A -85,B 0,C 180,E1 28088.409,E2 28088.409} C_VEL
LIN {X 0,Y 600.17,Z 1208.864,A -85,B 0,C 180,E1 28086.697,E2 28086.697} C_VEL
LIN {X 0,Y 600.036,Z 1214.097,A -85,B 0,C 180,E1 28084.971,E2 28084.971} C_VEL
LIN {X 0,Y 599.958,Z 1218.261,A -85,B 0,C 180,E1 28083.248,E2 28083.248} C_VEL
LIN {X 0,Y 599.917,Z 1221.402,A -85,B 0,C 180,E1 28081.528,E2 28081.528} C_VEL
LIN {X 0,Y 599.907,Z 1223.536,A -85,B 0,C 180,E1 28079.809,E2 28079.809} C_VEL
LIN {X 0,Y 599.913,Z 1224.677,A -85,B 0,C 180,E1 28078.09,E2 28078.09} C_VEL
LIN {X 0,Y 599.912,Z 1224.833,A -85,B 0,C 180,E1 28076.369,E2 28076.369} C_VEL
LIN {X 0,Y 599.911,Z 1224.01,A -85,B 0,C 180,E1 28074.644,E2 28074.644} C_VEL
LIN {X 0,Y 599.923,Z 1222.044,A -85,B 0,C 180,E1 28072.819,E2 28072.819} C_VEL
LIN {X 0,Y 599.945,Z 1219.133,A -85,B 0,C 180,E1 28071.083,E2 28071.083} C_VEL
LIN {X 0,Y 600.001,Z 1215.163,A -85,B 0,C 180,E1 28069.34,E2 28069.34} C_VEL
LIN {X 0,Y 600.137,Z 1210.099,A -85,B 0,C 180,E1 28067.589,E2 28067.589} C_VEL
LIN {X 0,Y 600.322,Z 1204.254,A -85,B 0,C 180,E1 28065.926,E2 28065.926} C_VEL
LIN {X 0,Y 600.634,Z 1197.058,A -85,B 0,C 180,E1 28064.2,E2 28064.2} C_VEL
LIN {X 0,Y 601.054,Z 1189.197,A -85,B 0,C 180,E1 28062.576,E2 28062.576} C_VEL
LIN {X 0,Y 601.616,Z 1180.55,A -85,B 0,C 180,E1 28060.989,E2 28060.989} C_VEL
LIN {X 0,Y 602.384,Z 1169.953,A -85,B 0,C 180,E1 28059.295,E2 28059.295} C_VEL
LIN {X 0,Y 603.356,Z 1157.691,A -85,B 0,C 180,E1 28057.594,E2 28057.594} C_VEL
LIN {X 0,Y 604.72,Z 1141.343,A -85,B 0,C 180,E1 28055.654,E2 28055.654} C_VEL
LIN {X 0,Y 606.052,Z 1125.581,A -85,B 0,C 180,E1 28054.05,E2 28054.05} C_VEL
LIN {X 0,Y 607.428,Z 1108.983,A -85,B 0,C 180,E1 28052.607,E2 28052.607} C_VEL
LIN {X 0,Y 608.818,Z 1091.515,A -85,B 0,C 180,E1 28051.285,E2 28051.285} C_VEL
LIN {X 0,Y 610.136,Z 1073.094,A -85,B 0,C 180,E1 28050.104,E2 28050.104} C_VEL
LIN {X 0,Y 611.507,Z 1051.993,A -85,B 0,C 180,E1 28048.961,E2 28048.961} C_VEL
LIN {X 0,Y 612.503,Z 1033.428,A -85,B 0,C 180,E1 28048.122,E2 28048.122} C_VEL
LIN {X 0,Y 613.471,Z 1011.636,A -85,B 0,C 180,E1 28047.323,E2 28047.323} C_VEL
LIN {X 0,Y 614.194,Z 990.099,A -85,B 0,C 180,E1 28046.699,E2 28046.699} C_VEL
LIN {X 0,Y 614.633,Z 968.044,A -85,B 0,C 180,E1 28046.242,E2 28046.242} C_VEL
LIN {X 0,Y 614.878,Z 942.383,A -85,B 0,C 180,E1 28045.889,E2 28045.889} C_VEL
LIN {X 0,Y 616.098,Z 777.912,A -85,B 0,C 180,E1 28043.998,E2 28043.998} C_VEL
LIN {X 0,Y 617.686,Z 656.482,A -85,B 0,C 180,E1 28042.447,E2 28042.447} C_VEL
LIN {X 0,Y 618.752,Z 655.84,A -85,B 0,C 180,E1 28042.291,E2 28042.291} C_VEL
LIN {X 0,Y 619.393,Z 657.833,A -85,B 0,C 180,E1 28041.218,E2 28041.218} C_VEL
LIN {X 0,Y 619.521,Z 658.557,A -85,B 0,C 180,E1 28040.967,E2 28040.967} C_VEL
LIN {X 0,Y 614.054,Z 668.961,A -85,B 0,C 180,E1 28039.647,E2 28039.647} C_VEL
LIN {X 0,Y 609.795,Z 681.246,A -85,B 0,C 180,E1 28038.323,E2 28038.323} C_VEL
LIN {X 0,Y 606.565,Z 696.006,A -85,B 0,C 180,E1 28036.964,E2 28036.964} C_VEL
LIN {X 0,Y 604.17,Z 714.423,A -85,B 0,C 180,E1 28035.505,E2 28035.505} C_VEL
LIN {X 0,Y 602.381,Z 739.324,A -85,B 0,C 180,E1 28033.775,E2 28033.775} C_VEL
LIN {X 0,Y 601.553,Z 774.072,A -85,B 0,C 180,E1 28031.584,E2 28031.584} C_VEL
LIN {X 0,Y 602.885,Z 795.305,A -85,B 0,C 180,E1 28030.278,E2 28030.278} C_VEL
LIN {X 0,Y 606.102,Z 814.59,A -85,B 0,C 180,E1 28029.087,E2 28029.087} C_VEL
LIN {X 0,Y 610.9,Z 831.024,A -85,B 0,C 180,E1 28028.068,E2 28028.068} C_VEL
LIN {X 0,Y 617.831,Z 847.114,A -85,B 0,C 180,E1 28027.073,E2 28027.073} C_VEL
LIN {X 0,Y 626.277,Z 861.548,A -85,B 0,C 180,E1 28026.19,E2 28026.19} C_VEL
LIN {X 0,Y 635.725,Z 874.044,A -85,B 0,C 180,E1 28025.439,E2 28025.439} C_VEL
LIN {X 0,Y 647.262,Z 886.173,A -85,B 0,C 180,E1 28024.731,E2 28024.731} C_VEL
LIN {X 0,Y 659.62,Z 896.676,A -85,B 0,C 180,E1 28024.141,E2 28024.141} C_VEL
LIN {X 0,Y 661.018,Z 897.953,A -85,B 0,C 180,E1 28024.071,E2 28024.071} C_VEL
LIN {X 0,Y 647.542,Z 909.657,A -85,B 0,C 180,E1 28023.454,E2 28023.454} C_VEL
LIN {X 0,Y 637.045,Z 921.029,A -85,B 0,C 180,E1 28022.84,E2 28022.84} C_VEL
LIN {X 0,Y 629.144,Z 932.17,A -85,B 0,C 180,E1 28022.223,E2 28022.223} C_VEL
LIN {X 0,Y 620.936,Z 945.902,A -85,B 0,C 180,E1 28021.47,E2 28021.47} C_VEL
LIN {X 0,Y 615.814,Z 964.391,A -85,B 0,C 180,E1 28021.416,E2 28021.416} C_VEL
LIN {X 0,Y 614.533,Z 975.532,A -85,B 0,C 180,E1 28021.323,E2 28021.323} C_VEL
LIN {X 0,Y 613.937,Z 1004.952,A -85,B 0,C 180,E1 28020.884,E2 28020.884} C_VEL
LIN {X 0,Y 612.916,Z 1033.832,A -85,B 0,C 180,E1 28020.281,E2 28020.281} C_VEL
LIN {X 0,Y 611.898,Z 1060.657,A -85,B 0,C 180,E1 28019.544,E2 28019.544} C_VEL
LIN {X 0,Y 610.856,Z 1086.121,A -85,B 0,C 180,E1 28018.674,E2 28018.674} C_VEL
LIN {X 0,Y 609.761,Z 1110.019,A -85,B 0,C 180,E1 28017.687,E2 28017.687} C_VEL
LIN {X 0,Y 608.679,Z 1132.066,A -85,B 0,C 180,E1 28016.607,E2 28016.607} C_VEL
LIN {X 0,Y 607.584,Z 1152.39,A -85,B 0,C 180,E1 28015.438,E2 28015.438} C_VEL
LIN {X 0,Y 606.343,Z 1174.066,A -85,B 0,C 180,E1 28013.995,E2 28013.995} C_VEL
LIN {X 0,Y 605.258,Z 1191.24,A -85,B 0,C 180,E1 28012.64,E2 28012.64} C_VEL
LIN {X 0,Y 604.378,Z 1205.157,A -85,B 0,C 180,E1 28011.396,E2 28011.396} C_VEL
LIN {X 0,Y 603.585,Z 1217.488,A -85,B 0,C 180,E1 28010.157,E2 28010.157} C_VEL
LIN {X 0,Y 602.865,Z 1228.858,A -85,B 0,C 180,E1 28008.871,E2 28008.871} C_VEL
LIN {X 0,Y 602.137,Z 1240.35,A -85,B 0,C 180,E1 28007.393,E2 28007.393} C_VEL
LIN {X 0,Y 601.549,Z 1250.38,A -85,B 0,C 180,E1 28005.919,E2 28005.919} C_VEL
LIN {X 0,Y 601.101,Z 1258.549,A -85,B 0,C 180,E1 28004.506,E2 28004.506} C_VEL
LIN {X 0,Y 600.644,Z 1266.902,A -85,B 0,C 180,E1 28002.793,E2 28002.793} C_VEL
LIN {X 0,Y 600.327,Z 1274.199,A -85,B 0,C 180,E1 28001.044,E2 28001.044} C_VEL
LIN {X 0,Y 600.122,Z 1280.306,A -85,B 0,C 180,E1 27999.302,E2 27999.302} C_VEL
LIN {X 0,Y 600.005,Z 1285.292,A -85,B 0,C 180,E1 27997.566,E2 27997.566} C_VEL
LIN {X 0,Y 599.929,Z 1289.431,A -85,B 0,C 180,E1 27995.724,E2 27995.724} C_VEL
LIN {X 0,Y 599.902,Z 1292.625,A -85,B 0,C 180,E1 27993.728,E2 27993.728} C_VEL
LIN {X 0,Y 599.896,Z 1294.64,A -85,B 0,C 180,E1 27991.338,E2 27991.338} C_VEL
LIN {X 0,Y 599.894,Z 1294.852,A -85,B 0,C 180,E1 27989.428,E2 27989.428} C_VEL
LIN {X 0,Y 599.899,Z 1293.955,A -85,B 0,C 180,E1 27987.613,E2 27987.613} C_VEL
LIN {X 0,Y 599.915,Z 1291.953,A -85,B 0,C 180,E1 27985.796,E2 27985.796} C_VEL
LIN {X 0,Y 599.936,Z 1289.02,A -85,B 0,C 180,E1 27984.07,E2 27984.07} C_VEL
LIN {X 0,Y 600.004,Z 1285.047,A -85,B 0,C 180,E1 27982.34,E2 27982.34} C_VEL
LIN {X 0,Y 600.136,Z 1280.005,A -85,B 0,C 180,E1 27980.604,E2 27980.604} C_VEL
LIN {X 0,Y 600.339,Z 1273.834,A -85,B 0,C 180,E1 27978.862,E2 27978.862} C_VEL
LIN {X 0,Y 600.643,Z 1266.904,A -85,B 0,C 180,E1 27977.21,E2 27977.21} C_VEL
LIN {X 0,Y 601.111,Z 1258.329,A -85,B 0,C 180,E1 27975.455,E2 27975.455} C_VEL
LIN {X 0,Y 601.584,Z 1249.842,A -85,B 0,C 180,E1 27973.985,E2 27973.985} C_VEL
LIN {X 0,Y 602.35,Z 1238.119,A -85,B 0,C 180,E1 27972.217,E2 27972.217} C_VEL
LIN {X 0,Y 603.402,Z 1222.826,A -85,B 0,C 180,E1 27970.244,E2 27970.244} C_VEL
LIN {X 0,Y 604.471,Z 1208.429,A -85,B 0,C 180,E1 27968.638,E2 27968.638} C_VEL
LIN {X 0,Y 605.623,Z 1193.574,A -85,B 0,C 180,E1 27967.172,E2 27967.172} C_VEL
LIN {X 0,Y 607.007,Z 1176.486,A -85,B 0,C 180,E1 27965.683,E2 27965.683} C_VEL
LIN {X 0,Y 608.655,Z 1156.103,A -85,B 0,C 180,E1 27964.143,E2 27964.143} C_VEL
LIN {X 0,Y 610.325,Z 1135.37,A -85,B 0,C 180,E1 27962.803,E2 27962.803} C_VEL
LIN {X 0,Y 612.075,Z 1113.047,A -85,B 0,C 180,E1 27961.565,E2 27961.565} C_VEL
LIN {X 0,Y 613.786,Z 1090.889,A -85,B 0,C 180,E1 27960.532,E2 27960.532} C_VEL
LIN {X 0,Y 615.432,Z 1067.337,A -85,B 0,C 180,E1 27959.623,E2 27959.623} C_VEL
LIN {X 0,Y 617.091,Z 1042.944,A -85,B 0,C 180,E1 27958.872,E2 27958.872} C_VEL
LIN {X 0,Y 618.429,Z 1019.021,A -85,B 0,C 180,E1 27958.319,E2 27958.319} C_VEL
LIN {X 0,Y 619.44,Z 993.353,A -85,B 0,C 180,E1 27957.895,E2 27957.895} C_VEL
LIN {X 0,Y 620.275,Z 970.32,A -85,B 0,C 180,E1 27957.599,E2 27957.599} C_VEL
LIN {X 0,Y 621.206,Z 963.618,A -85,B 0,C 180,E1 27957.536,E2 27957.536} C_VEL
LIN {X 0,Y 626.839,Z 952.527,A -85,B 0,C 180,E1 27956.941,E2 27956.941} C_VEL
LIN {X 0,Y 637.952,Z 934.556,A -85,B 0,C 180,E1 27956.086,E2 27956.086} C_VEL
LIN {X 0,Y 646.915,Z 922.877,A -85,B 0,C 180,E1 27955.626,E2 27955.626} C_VEL
LIN {X 0,Y 658.919,Z 909.756,A -85,B 0,C 180,E1 27955.212,E2 27955.212} C_VEL
LIN {X 0,Y 663.593,Z 904.928,A -85,B 0,C 180,E1 27955.075,E2 27955.075} C_VEL
LIN {X 0,Y 652.4,Z 898.104,A -85,B 0,C 180,E1 27954.021,E2 27954.021} C_VEL
LIN {X 0,Y 642.906,Z 890.227,A -85,B 0,C 180,E1 27952.926,E2 27952.926} C_VEL
LIN {X 0,Y 634.469,Z 880.612,A -85,B 0,C 180,E1 27951.705,E2 27951.705} C_VEL
LIN {X 0,Y 627.693,Z 869.479,A -85,B 0,C 180,E1 27950.42,E2 27950.42} C_VEL
LIN {X 0,Y 622.622,Z 856.776,A -85,B 0,C 180,E1 27949.066,E2 27949.066} C_VEL
LIN {X 0,Y 619.448,Z 842.735,A -85,B 0,C 180,E1 27947.695,E2 27947.695} C_VEL
LIN {X 0,Y 618.171,Z 826.508,A -85,B 0,C 180,E1 27946.231,E2 27946.231} C_VEL
LIN {X 0,Y 619.073,Z 803.636,A -85,B 0,C 180,E1 27944.318,E2 27944.318} C_VEL
LIN {X 0,Y 621.706,Z 766.827,A -85,B 0,C 180,E1 27941.255,E2 27941.255} C_VEL
LIN {X 0,Y 624.23,Z 731.565,A -85,B 0,C 180,E1 27938.25,E2 27938.25} C_VEL
LIN {X 0,Y 626.634,Z 698.345,A -85,B 0,C 180,E1 27935.34,E2 27935.34} C_VEL
LIN {X 0,Y 628.246,Z 675.198,A -85,B 0,C 180,E1 27933.25,E2 27933.25} C_VEL
LIN {X 0,Y 619.837,Z 655.258,A -85,B 0,C 180,E1 27930.433,E2 27930.433} C_VEL
LIN {X 0,Y 612.068,Z 637.451,A -85,B 0,C 180,E1 27927.748,E2 27927.748} C_VEL
LIN {X 0,Y 605.95,Z 624.253,A -85,B 0,C 180,E1 27925.616,E2 27925.616} C_VEL
LIN {X 0,Y 602.652,Z 616.881,A -85,B 0,C 180,E1 27924.402,E2 27924.402} C_VEL
LIN {X 0,Y 601.177,Z 613.49,A -85,B 0,C 180,E1 27923.832,E2 27923.832} C_VEL
LIN {X 0,Y 601.122,Z 613.103,A -85,B 0,C 180,E1 27923.737,E2 27923.737} C_VEL
LIN {X 0,Y 601.131,Z 613.099,A -85,B 0,C 180,E1 27920.54,E2 27920.54} C_VEL
LIN {X 0,Y 601.132,Z 613.097,A -85,B 0,C 180,E1 27917.222,E2 27917.222} C_VEL
LIN {X 0,Y 601.135,Z 613.101,A -85,B 0,C 180,E1 27913.858,E2 27913.858} C_VEL
LIN {X 0,Y 601.123,Z 613.096,A -85,B 0,C 180,E1 27910.64,E2 27910.64} C_VEL
LIN {X 0,Y 601.123,Z 613.101,A -85,B 0,C 180,E1 27907.455,E2 27907.455} C_VEL
LIN {X 0,Y 601.119,Z 613.102,A -85,B 0,C 180,E1 27904.293,E2 27904.293} C_VEL
LIN {X 0,Y 601.119,Z 613.097,A -85,B 0,C 180,E1 27901.144,E2 27901.144} C_VEL
LIN {X 0,Y 601.118,Z 613.098,A -85,B 0,C 180,E1 27897.998,E2 27897.998} C_VEL
LIN {X 0,Y 601.118,Z 613.1,A -85,B 0,C 180,E1 27894.847,E2 27894.847} C_VEL
LIN {X 0,Y 601.12,Z 613.101,A -85,B 0,C 180,E1 27891.759,E2 27891.759} C_VEL
LIN {X 0,Y 601.119,Z 613.101,A -85,B 0,C 180,E1 27888.583,E2 27888.583} C_VEL
LIN {X 0,Y 601.118,Z 613.102,A -85,B 0,C 180,E1 27885.453,E2 27885.453} C_VEL
LIN {X 0,Y 601.12,Z 613.101,A -85,B 0,C 180,E1 27882.278,E2 27882.278} C_VEL
LIN {X 0,Y 601.119,Z 613.1,A -85,B 0,C 180,E1 27879.147,E2 27879.147} C_VEL
LIN {X 0,Y 601.118,Z 613.098,A -85,B 0,C 180,E1 27876.054,E2 27876.054} C_VEL
LIN {X 0,Y 601.119,Z 613.094,A -85,B 0,C 180,E1 27872.886,E2 27872.886} C_VEL
LIN {X 0,Y 601.121,Z 613.097,A -85,B 0,C 180,E1 27869.735,E2 27869.735} C_VEL
LIN {X 0,Y 601.126,Z 613.1,A -85,B 0,C 180,E1 27866.593,E2 27866.593} C_VEL
LIN {X 0,Y 601.125,Z 613.101,A -85,B 0,C 180,E1 27863.334,E2 27863.334} C_VEL
LIN {X 0,Y 601.138,Z 613.099,A -85,B 0,C 180,E1 27860.055,E2 27860.055} C_VEL
LIN {X 0,Y 601.128,Z 613.077,A -85,B 0,C 180,E1 27856.74,E2 27856.74} C_VEL
LIN {X 0,Y 601.133,Z 613.1,A -85,B 0,C 180,E1 27853.513,E2 27853.513} C_VEL
LIN {X 0,Y 601.126,Z 613.1,A -85,B 0,C 180,E1 27850.317,E2 27850.317} C_VEL
LIN {X 0,Y 601.125,Z 613.092,A -85,B 0,C 180,E1 27847.14,E2 27847.14} C_VEL
LIN {X 0,Y 601.121,Z 613.092,A -85,B 0,C 180,E1 27843.977,E2 27843.977} C_VEL
LIN {X 0,Y 601.13,Z 613.152,A -85,B 0,C 180,E1 27843.582,E2 27843.582} C_VEL
LIN {X 0,Y 609.774,Z 640.125,A -85,B 0,C 180,E1 27841.315,E2 27841.315} C_VEL
LIN {X 0,Y 610.905,Z 644.966,A -85,B 0,C 180,E1 27840.924,E2 27840.924} C_VEL
LIN {X 0,Y 610.881,Z 646.149,A -85,B 0,C 180,E1 27840.844,E2 27840.844} C_VEL
LIN {X 0,Y 609.833,Z 652.598,A -85,B 0,C 180,E1 27840.449,E2 27840.449} C_VEL
LIN {X 0,Y 603.672,Z 670.302,A -85,B 0,C 180,E1 27839.501,E2 27839.501} C_VEL
LIN {X 0,Y 602.85,Z 675.783,A -85,B 0,C 180,E1 27839.149,E2 27839.149} C_VEL
LIN {X 0,Y 601.542,Z 717.519,A -85,B 0,C 180,E1 27836.206,E2 27836.206} C_VEL
LIN {X 0,Y 600.07,Z 762.12,A -85,B 0,C 180,E1 27833.051,E2 27833.051} C_VEL
LIN {X 0,Y 598.733,Z 809.781,A -85,B 0,C 180,E1 27829.764,E2 27829.764} C_VEL
LIN {X 0,Y 598.225,Z 840.586,A -85,B 0,C 180,E1 27827.749,E2 27827.749} C_VEL
LIN {X 0,Y 599.006,Z 849.101,A -85,B 0,C 180,E1 27827.617,E2 27827.617} C_VEL
LIN {X 0,Y 597.639,Z 1010.198,A -85,B 0,C 180,E1 27825.637,E2 27825.637} C_VEL
LIN {X 0,Y 597.419,Z 1027.639,A -85,B 0,C 180,E1 27825.245,E2 27825.245} C_VEL
LIN {X 0,Y 597.026,Z 1044.009,A -85,B 0,C 180,E1 27824.697,E2 27824.697} C_VEL
LIN {X 0,Y 596.494,Z 1060.228,A -85,B 0,C 180,E1 27823.967,E2 27823.967} C_VEL
LIN {X 0,Y 595.883,Z 1075.393,A -85,B 0,C 180,E1 27823.091,E2 27823.091} C_VEL
LIN {X 0,Y 595.229,Z 1089.476,A -85,B 0,C 180,E1 27822.07,E2 27822.07} C_VEL
LIN {X 0,Y 594.594,Z 1101.993,A -85,B 0,C 180,E1 27820.953,E2 27820.953} C_VEL
LIN {X 0,Y 593.987,Z 1113.584,A -85,B 0,C 180,E1 27819.69,E2 27819.69} C_VEL
LIN {X 0,Y 593.47,Z 1123.75,A -85,B 0,C 180,E1 27818.33,E2 27818.33} C_VEL
LIN {X 0,Y 593.052,Z 1132.494,A -85,B 0,C 180,E1 27816.874,E2 27816.874} C_VEL
LIN {X 0,Y 592.739,Z 1139.754,A -85,B 0,C 180,E1 27815.322,E2 27815.322} C_VEL
LIN {X 0,Y 592.532,Z 1145.509,A -85,B 0,C 180,E1 27813.675,E2 27813.675} C_VEL
LIN {X 0,Y 592.411,Z 1149.456,A -85,B 0,C 180,E1 27812.03,E2 27812.03} C_VEL
LIN {X 0,Y 592.356,Z 1151.754,A -85,B 0,C 180,E1 27810.289,E2 27810.289} C_VEL
LIN {X 0,Y 592.34,Z 1152.232,A -85,B 0,C 180,E1 27808.548,E2 27808.548} C_VEL
LIN {X 0,Y 592.376,Z 1150.933,A -85,B 0,C 180,E1 27806.806,E2 27806.806} C_VEL
LIN {X 0,Y 592.462,Z 1147.99,A -85,B 0,C 180,E1 27805.158,E2 27805.158} C_VEL
LIN {X 0,Y 592.623,Z 1143.252,A -85,B 0,C 180,E1 27803.508,E2 27803.508} C_VEL
LIN {X 0,Y 592.879,Z 1136.627,A -85,B 0,C 180,E1 27801.855,E2 27801.855} C_VEL
LIN {X 0,Y 593.263,Z 1128.414,A -85,B 0,C 180,E1 27800.296,E2 27800.296} C_VEL
LIN {X 0,Y 593.753,Z 1118.548,A -85,B 0,C 180,E1 27798.832,E2 27798.832} C_VEL
LIN {X 0,Y 594.361,Z 1107.116,A -85,B 0,C 180,E1 27797.465,E2 27797.465} C_VEL
LIN {X 0,Y 595.03,Z 1094.437,A -85,B 0,C 180,E1 27796.235,E2 27796.235} C_VEL
LIN {X 0,Y 595.687,Z 1080.799,A -85,B 0,C 180,E1 27795.167,E2 27795.167} C_VEL
LIN {X 0,Y 596.358,Z 1065.219,A -85,B 0,C 180,E1 27794.188,E2 27794.188} C_VEL
LIN {X 0,Y 596.935,Z 1049.28,A -85,B 0,C 180,E1 27793.405,E2 27793.405} C_VEL
LIN {X 0,Y 597.377,Z 1032.413,A -85,B 0,C 180,E1 27792.788,E2 27792.788} C_VEL
LIN {X 0,Y 597.664,Z 1014.376,A -85,B 0,C 180,E1 27792.33,E2 27792.33} C_VEL
LIN {X 0,Y 597.801,Z 993.821,A -85,B 0,C 180,E1 27792.027,E2 27792.027} C_VEL
LIN {X 0,Y 598.906,Z 844.974,A -85,B 0,C 180,E1 27790.21,E2 27790.21} C_VEL
LIN {X 0,Y 598.242,Z 839.673,A -85,B 0,C 180,E1 27790.1,E2 27790.1} C_VEL
LIN {X 0,Y 599.306,Z 792.279,A -85,B 0,C 180,E1 27786.915,E2 27786.915} C_VEL
LIN {X 0,Y 600.772,Z 746.017,A -85,B 0,C 180,E1 27783.669,E2 27783.669} C_VEL
LIN {X 0,Y 602.25,Z 703.11,A -85,B 0,C 180,E1 27780.617,E2 27780.617} C_VEL
LIN {X 0,Y 603.527,Z 661.27,A -85,B 0,C 180,E1 27777.666,E2 27777.666} C_VEL
LIN {X 0,Y 603.727,Z 646.595,A -85,B 0,C 180,E1 27776.642,E2 27776.642} C_VEL
LIN {X 0,Y 595.95,Z 622.208,A -85,B 0,C 180,E1 27774.538,E2 27774.538} C_VEL
LIN {X 0,Y 593.186,Z 614.076,A -85,B 0,C 180,E1 27773.817,E2 27773.817} C_VEL
LIN {X 0,Y 593.201,Z 614.07,A -85,B 0,C 180,E1 27770.534,E2 27770.534} C_VEL
LIN {X 0,Y 593.198,Z 614.088,A -85,B 0,C 180,E1 27767.211,E2 27767.211} C_VEL
LIN {X 0,Y 593.19,Z 614.088,A -85,B 0,C 180,E1 27763.964,E2 27763.964} C_VEL
LIN {X 0,Y 593.183,Z 614.088,A -85,B 0,C 180,E1 27760.719,E2 27760.719} C_VEL
LIN {X 0,Y 593.2,Z 614.092,A -85,B 0,C 180,E1 27757.603,E2 27757.603} C_VEL
LIN {X 0,Y 593.204,Z 614.233,A -85,B 0,C 180,E1 27756.224,E2 27756.224} C_VEL
LIN {X 0,Y 594.317,Z 617.28,A -85,B 0,C 180,E1 27755.813,E2 27755.813} C_VEL
LIN {X 0,Y 596.877,Z 623.005,A -85,B 0,C 180,E1 27755.039,E2 27755.039} C_VEL
LIN {X 0,Y 614.239,Z 648.698,A -85,B 0,C 180,E1 27753.31,E2 27753.31} C_VEL
LIN {X 0,Y 617.833,Z 655.108,A -85,B 0,C 180,E1 27752.957,E2 27752.957} C_VEL
LIN {X 0,Y 611.92,Z 892.402,A -85,B 0,C 180,E1 27749.657,E2 27749.657} C_VEL
LIN {X 0,Y 610.548,Z 957.631,A -85,B 0,C 180,E1 27748.749,E2 27748.749} C_VEL
LIN {X 0,Y 609.668,Z 980.753,A -85,B 0,C 180,E1 27748.251,E2 27748.251} C_VEL
LIN {X 0,Y 608.504,Z 1004.634,A -85,B 0,C 180,E1 27747.553,E2 27747.553} C_VEL
